LIN {X 0,Y 162.657,Z 541.681,A -85,B 0,C 180,E1 -31313.823,E2 -31313.823} C_VEL
LIN {X 0,Y 162.251,Z 555.226,A -85,B 0,C 180,E1 -31317.216,E2 -31317.216} C_VEL
LIN {X 0,Y 162.332,Z 566.74,A -85,B 0,C 180,E1 -31320.617,E2 -31320.617} C_VEL
LIN {X 0,Y 162.635,Z 577.197,A -85,B 0,C 180,E1 -31324.322,E2 -31324.322} C_VEL
LIN {X 0,Y 163.981,Z 589.038,A -85,B 0,C 180,E1 -31329.217,E2 -31329.217} C_VEL
LIN {X 0,Y 166.282,Z 597.77,A -85,B 0,C 180,E1 -31333.396,E2 -31333.396} C_VEL
LIN {X 0,Y 169.959,Z 606.171,A -85,B 0,C 180,E1 -31338.004,E2 -31338.004} C_VEL
LIN {X 0,Y 174.987,Z 613.199,A -85,B 0,C 180,E1 -31342.35,E2 -31342.35} C_VEL
LIN {X 0,Y 181.432,Z 619.004,A -85,B 0,C 180,E1 -31346.357,E2 -31346.357} C_VEL
LIN {X 0,Y 187.096,Z 622.568,A -85,B 0,C 180,E1 -31349.123,E2 -31349.123} C_VEL
LIN {X 0,Y 195.33,Z 626.257,A -85,B 0,C 180,E1 -31352.54,E2 -31352.54} C_VEL
LIN {X 0,Y 204.429,Z 628.796,A -85,B 0,C 180,E1 -31355.625,E2 -31355.625} C_VEL
LIN {X 0,Y 215.008,Z 630.267,A -85,B 0,C 180,E1 -31358.568,E2 -31358.568} C_VEL
LIN {X 0,Y 224.82,Z 630.463,A -85,B 0,C 180,E1 -31360.864,E2 -31360.864} C_VEL
LIN {X 0,Y 223.785,Z 630.854,A -85,B 0,C 180,E1 -31361.305,E2 -31361.305} C_VEL
LIN {X 0,Y 212.898,Z 633.183,A -85,B 0,C 180,E1 -31363.629,E2 -31363.629} C_VEL
LIN {X 0,Y 202.784,Z 634.608,A -85,B 0,C 180,E1 -31366.304,E2 -31366.304} C_VEL
LIN {X 0,Y 191.702,Z 635.182,A -85,B 0,C 180,E1 -31370.112,E2 -31370.112} C_VEL
LIN {X 0,Y 181.866,Z 634.463,A -85,B 0,C 180,E1 -31374.709,E2 -31374.709} C_VEL
LIN {X 0,Y 174.373,Z 632.741,A -85,B 0,C 180,E1 -31379.693,E2 -31379.693} C_VEL
LIN {X 0,Y 169.565,Z 638.187,A -85,B 0,C 180,E1 -31382.974,E2 -31382.974} C_VEL
LIN {X 0,Y 165.423,Z 642.984,A -85,B 0,C 180,E1 -31386.802,E2 -31386.802} C_VEL
LIN {X 0,Y 162.986,Z 645.969,A -85,B 0,C 180,E1 -31389.891,E2 -31389.891} C_VEL
LIN {X 0,Y 160.488,Z 649.343,A -85,B 0,C 180,E1 -31394.819,E2 -31394.819} C_VEL
LIN {X 0,Y 159.934,Z 650.447,A -85,B 0,C 180,E1 -31397.145,E2 -31397.145} C_VEL
LIN {X 0,Y 159.044,Z 651.219,A -85,B 0,C 180,E1 -31399.228,E2 -31399.228} C_VEL
LIN {X 0,Y 156.456,Z 651.707,A -85,B 0,C 180,E1 -31402.706,E2 -31402.706} C_VEL
LIN {X 0,Y 154.735,Z 651.565,A -85,B 0,C 180,E1 -31406.289,E2 -31406.289} C_VEL
LIN {X 0,Y 155.199,Z 651.263,A -85,B 0,C 180,E1 -31408.455,E2 -31408.455} C_VEL
LIN {X 0,Y 157.81,Z 650.765,A -85,B 0,C 180,E1 -31411.987,E2 -31411.987} C_VEL
LIN {X 0,Y 157.787,Z 658.681,A -85,B 0,C 180,E1 -31415.093,E2 -31415.093} C_VEL
LIN {X 0,Y 157.477,Z 665.759,A -85,B 0,C 180,E1 -31418.522,E2 -31418.522} C_VEL
LIN {X 0,Y 157.557,Z 673.281,A -85,B 0,C 180,E1 -31422.843,E2 -31422.843} C_VEL
LIN {X 0,Y 158.912,Z 680.871,A -85,B 0,C 180,E1 -31427.971,E2 -31427.971} C_VEL
LIN {X 0,Y 161.869,Z 687.258,A -85,B 0,C 180,E1 -31432.92,E2 -31432.92} C_VEL
LIN {X 0,Y 166.542,Z 692.636,A -85,B 0,C 180,E1 -31437.557,E2 -31437.557} C_VEL
LIN {X 0,Y 172.573,Z 696.952,A -85,B 0,C 180,E1 -31441.846,E2 -31441.846} C_VEL
LIN {X 0,Y 179.734,Z 700.291,A -85,B 0,C 180,E1 -31445.772,E2 -31445.772} C_VEL
LIN {X 0,Y 188.2,Z 702.78,A -85,B 0,C 180,E1 -31449.25,E2 -31449.25} C_VEL
LIN {X 0,Y 197.682,Z 704.359,A -85,B 0,C 180,E1 -31452.316,E2 -31452.316} C_VEL
LIN {X 0,Y 207.92,Z 704.957,A -85,B 0,C 180,E1 -31455.028,E2 -31455.028} C_VEL
LIN {X 0,Y 197.945,Z 704.33,A -85,B 0,C 180,E1 -31457.753,E2 -31457.753} C_VEL
LIN {X 0,Y 188.578,Z 702.73,A -85,B 0,C 180,E1 -31460.844,E2 -31460.844} C_VEL
LIN {X 0,Y 180.062,Z 700.21,A -85,B 0,C 180,E1 -31464.303,E2 -31464.303} C_VEL
LIN {X 0,Y 172.782,Z 696.814,A -85,B 0,C 180,E1 -31468.197,E2 -31468.197} C_VEL
LIN {X 0,Y 165.469,Z 691.187,A -85,B 0,C 180,E1 -31473.611,E2 -31473.611} C_VEL
LIN {X 0,Y 161.091,Z 685.52,A -85,B 0,C 180,E1 -31478.31,E2 -31478.31} C_VEL
LIN {X 0,Y 158.325,Z 678.763,A -85,B 0,C 180,E1 -31483.288,E2 -31483.288} C_VEL
LIN {X 0,Y 157.225,Z 669.662,A -85,B 0,C 180,E1 -31489.086,E2 -31489.086} C_VEL
LIN {X 0,Y 157.41,Z 661.083,A -85,B 0,C 180,E1 -31493.614,E2 -31493.614} C_VEL
LIN {X 0,Y 157.623,Z 653.684,A -85,B 0,C 180,E1 -31496.816,E2 -31496.816} C_VEL
LIN {X 0,Y 157.444,Z 644.543,A -85,B 0,C 180,E1 -31500.001,E2 -31500.001} C_VEL
LIN {X 0,Y 157.364,Z 633.619,A -85,B 0,C 180,E1 -31503.19,E2 -31503.19} C_VEL
LIN {X 0,Y 157.453,Z 620.345,A -85,B 0,C 180,E1 -31506.386,E2 -31506.386} C_VEL
LIN {X 0,Y 157.743,Z 605.275,A -85,B 0,C 180,E1 -31509.264,E2 -31509.264} C_VEL
LIN {X 0,Y 158.123,Z 591.449,A -85,B 0,C 180,E1 -31511.364,E2 -31511.364} C_VEL
LIN {X 0,Y 158.427,Z 575.605,A -85,B 0,C 180,E1 -31513.178,E2 -31513.178} C_VEL
LIN {X 0,Y 159.069,Z 531.92,A -85,B 0,C 180,E1 -31517.292,E2 -31517.292} C_VEL
LIN {X 0,Y 160.564,Z 481.479,A -85,B 0,C 180,E1 -31521.892,E2 -31521.892} C_VEL
LIN {X 0,Y 158.603,Z 451.78,A -85,B 0,C 180,E1 -31524.372,E2 -31524.372} C_VEL
LIN {X 0,Y 158.469,Z 439.257,A -85,B 0,C 180,E1 -31525.529,E2 -31525.529} C_VEL
LIN {X 0,Y 161.863,Z 413.266,A -85,B 0,C 180,E1 -31532.747,E2 -31532.747} C_VEL
LIN {X 0,Y 160.879,Z 408.168,A -85,B 0,C 180,E1 -31534.185,E2 -31534.185} C_VEL
LIN {X 0,Y 161.476,Z 409.866,A -85,B 0,C 180,E1 -31534.704,E2 -31534.704} C_VEL
LIN {X 0,Y 162.33,Z 410.505,A -85,B 0,C 180,E1 -31535.249,E2 -31535.249} C_VEL
LIN {X 0,Y 164.016,Z 410.046,A -85,B 0,C 180,E1 -31536.149,E2 -31536.149} C_VEL
LIN {X 0,Y 165.523,Z 408.754,A -85,B 0,C 180,E1 -31536.852,E2 -31536.852} C_VEL
LIN {X 0,Y 169.339,Z 408.335,A -85,B 0,C 180,E1 -31538.729,E2 -31538.729} C_VEL
LIN {X 0,Y 171.509,Z 407.086,A -85,B 0,C 180,E1 -31539.653,E2 -31539.653} C_VEL
LIN {X 0,Y 175.345,Z 406.759,A -85,B 0,C 180,E1 -31541.309,E2 -31541.309} C_VEL
LIN {X 0,Y 180.627,Z 415.01,A -85,B 0,C 180,E1 -31543.911,E2 -31543.911} C_VEL
LIN {X 0,Y 186.581,Z 425.308,A -85,B 0,C 180,E1 -31546.581,E2 -31546.581} C_VEL
LIN {X 0,Y 192.729,Z 437.493,A -85,B 0,C 180,E1 -31549.124,E2 -31549.124} C_VEL
LIN {X 0,Y 194.185,Z 440.713,A -85,B 0,C 180,E1 -31549.703,E2 -31549.703} C_VEL
LIN {X 0,Y 191.472,Z 490.951,A -85,B 0,C 180,E1 -31551.492,E2 -31551.492} C_VEL
LIN {X 0,Y 190.329,Z 504.695,A -85,B 0,C 180,E1 -31552.278,E2 -31552.278} C_VEL
LIN {X 0,Y 188.23,Z 519.107,A -85,B 0,C 180,E1 -31553.46,E2 -31553.46} C_VEL
LIN {X 0,Y 185.58,Z 531.813,A -85,B 0,C 180,E1 -31554.859,E2 -31554.859} C_VEL
LIN {X 0,Y 182.689,Z 543.452,A -85,B 0,C 180,E1 -31556.554,E2 -31556.554} C_VEL
LIN {X 0,Y 179.123,Z 555.581,A -85,B 0,C 180,E1 -31558.793,E2 -31558.793} C_VEL
LIN {X 0,Y 175.219,Z 566.598,A -85,B 0,C 180,E1 -31561.334,E2 -31561.334} C_VEL
LIN {X 0,Y 170.85,Z 577.269,A -85,B 0,C 180,E1 -31564.434,E2 -31564.434} C_VEL
LIN {X 0,Y 166.886,Z 586.379,A -85,B 0,C 180,E1 -31567.806,E2 -31567.806} C_VEL
LIN {X 0,Y 163.004,Z 594.923,A -85,B 0,C 180,E1 -31571.848,E2 -31571.848} C_VEL
LIN {X 0,Y 159.652,Z 601.853,A -85,B 0,C 180,E1 -31576.037,E2 -31576.037} C_VEL
LIN {X 0,Y 156.764,Z 608.082,A -85,B 0,C 180,E1 -31581.003,E2 -31581.003} C_VEL
LIN {X 0,Y 155.173,Z 611.678,A -85,B 0,C 180,E1 -31584.821,E2 -31584.821} C_VEL
LIN {X 0,Y 154.059,Z 615.204,A -85,B 0,C 180,E1 -31590,E2 -31590} C_VEL
LIN {X 0,Y 153.894,Z 617.381,A -85,B 0,C 180,E1 -31595.223,E2 -31595.223} C_VEL
LIN {X 0,Y 154.588,Z 618.271,A -85,B 0,C 180,E1 -31600.443,E2 -31600.443} C_VEL
LIN {X 0,Y 156.181,Z 617.88,A -85,B 0,C 180,E1 -31605.611,E2 -31605.611} C_VEL
LIN {X 0,Y 158.917,Z 616.168,A -85,B 0,C 180,E1 -31610.648,E2 -31610.648} C_VEL
LIN {X 0,Y 162.647,Z 613.091,A -85,B 0,C 180,E1 -31615.51,E2 -31615.51} C_VEL
LIN {X 0,Y 167.258,Z 608.524,A -85,B 0,C 180,E1 -31620.169,E2 -31620.169} C_VEL
LIN {X 0,Y 172.76,Z 602.335,A -85,B 0,C 180,E1 -31624.585,E2 -31624.585} C_VEL
LIN {X 0,Y 177.961,Z 595.766,A -85,B 0,C 180,E1 -31628.075,E2 -31628.075} C_VEL
LIN {X 0,Y 183.455,Z 588.119,A -85,B 0,C 180,E1 -31631.195,E2 -31631.195} C_VEL
LIN {X 0,Y 189.122,Z 579.325,A -85,B 0,C 180,E1 -31633.983,E2 -31633.983} C_VEL
LIN {X 0,Y 194.653,Z 569.152,A -85,B 0,C 180,E1 -31636.583,E2 -31636.583} C_VEL
LIN {X 0,Y 200.076,Z 557.787,A -85,B 0,C 180,E1 -31638.825,E2 -31638.825} C_VEL
LIN {X 0,Y 204.966,Z 545.823,A -85,B 0,C 180,E1 -31640.641,E2 -31640.641} C_VEL
LIN {X 0,Y 208.697,Z 534.273,A -85,B 0,C 180,E1 -31642.067,E2 -31642.067} C_VEL
LIN {X 0,Y 212.105,Z 520.79,A -85,B 0,C 180,E1 -31643.373,E2 -31643.373} C_VEL
LIN {X 0,Y 214.577,Z 507.153,A -85,B 0,C 180,E1 -31644.357,E2 -31644.357} C_VEL
LIN {X 0,Y 216.23,Z 493.322,A -85,B 0,C 180,E1 -31645.033,E2 -31645.033} C_VEL
LIN {X 0,Y 218.184,Z 463.682,A -85,B 0,C 180,E1 -31646.002,E2 -31646.002} C_VEL
LIN {X 0,Y 212.944,Z 453.225,A -85,B 0,C 180,E1 -31648.622,E2 -31648.622} C_VEL
LIN {X 0,Y 210.989,Z 449.575,A -85,B 0,C 180,E1 -31649.667,E2 -31649.667} C_VEL
LIN {X 0,Y 206.99,Z 459.803,A -85,B 0,C 180,E1 -31650.788,E2 -31650.788} C_VEL
LIN {X 0,Y 203.4,Z 466.877,A -85,B 0,C 180,E1 -31652.013,E2 -31652.013} C_VEL
LIN {X 0,Y 202.486,Z 468.575,A -85,B 0,C 180,E1 -31652.347,E2 -31652.347} C_VEL
LIN {X 0,Y 198.679,Z 481.103,A -85,B 0,C 180,E1 -31653.401,E2 -31653.401} C_VEL
LIN {X 0,Y 195.565,Z 489.455,A -85,B 0,C 180,E1 -31654.47,E2 -31654.47} C_VEL
LIN {X 0,Y 192.222,Z 496.043,A -85,B 0,C 180,E1 -31655.863,E2 -31655.863} C_VEL
LIN {X 0,Y 191.222,Z 497.747,A -85,B 0,C 180,E1 -31656.313,E2 -31656.313} C_VEL
LIN {X 0,Y 187.469,Z 508.563,A -85,B 0,C 180,E1 -31657.322,E2 -31657.322} C_VEL
LIN {X 0,Y 184.183,Z 515.642,A -85,B 0,C 180,E1 -31658.308,E2 -31658.308} C_VEL
LIN {X 0,Y 180.852,Z 521.347,A -85,B 0,C 180,E1 -31659.525,E2 -31659.525} C_VEL
LIN {X 0,Y 178.031,Z 525.18,A -85,B 0,C 180,E1 -31660.781,E2 -31660.781} C_VEL
LIN {X 0,Y 175.796,Z 527.75,A -85,B 0,C 180,E1 -31662.013,E2 -31662.013} C_VEL
LIN {X 0,Y 171.998,Z 533.916,A -85,B 0,C 180,E1 -31663.436,E2 -31663.436} C_VEL
LIN {X 0,Y 168.996,Z 537.903,A -85,B 0,C 180,E1 -31664.986,E2 -31664.986} C_VEL
LIN {X 0,Y 168.114,Z 538.939,A -85,B 0,C 180,E1 -31665.522,E2 -31665.522} C_VEL
LIN {X 0,Y 166.791,Z 540.084,A -85,B 0,C 180,E1 -31666.645,E2 -31666.645} C_VEL
LIN {X 0,Y 165.194,Z 542.014,A -85,B 0,C 180,E1 -31667.759,E2 -31667.759} C_VEL
LIN {X 0,Y 162.353,Z 546.074,A -85,B 0,C 180,E1 -31669.371,E2 -31669.371} C_VEL
LIN {X 0,Y 161.493,Z 547.163,A -85,B 0,C 180,E1 -31670.008,E2 -31670.008} C_VEL
LIN {X 0,Y 160.015,Z 548.819,A -85,B 0,C 180,E1 -31671.509,E2 -31671.509} C_VEL
LIN {X 0,Y 159.456,Z 549.259,A -85,B 0,C 180,E1 -31672.427,E2 -31672.427} C_VEL
LIN {X 0,Y 158.404,Z 550.699,A -85,B 0,C 180,E1 -31673.472,E2 -31673.472} C_VEL
LIN {X 0,Y 156.612,Z 553.438,A -85,B 0,C 180,E1 -31674.867,E2 -31674.867} C_VEL
LIN {X 0,Y 155.163,Z 555.396,A -85,B 0,C 180,E1 -31677.412,E2 -31677.412} C_VEL
LIN {X 0,Y 155.611,Z 554.521,A -85,B 0,C 180,E1 -31678.145,E2 -31678.145} C_VEL
LIN {X 0,Y 155.791,Z 566.718,A -85,B 0,C 180,E1 -31681.932,E2 -31681.932} C_VEL
LIN {X 0,Y 156.222,Z 577.22,A -85,B 0,C 180,E1 -31685.789,E2 -31685.789} C_VEL
LIN {X 0,Y 157.591,Z 587.719,A -85,B 0,C 180,E1 -31690.24,E2 -31690.24} C_VEL
LIN {X 0,Y 160.433,Z 597.884,A -85,B 0,C 180,E1 -31695.186,E2 -31695.186} C_VEL
LIN {X 0,Y 164.519,Z 606.427,A -85,B 0,C 180,E1 -31699.913,E2 -31699.913} C_VEL
LIN {X 0,Y 170.034,Z 613.597,A -85,B 0,C 180,E1 -31704.326,E2 -31704.326} C_VEL
LIN {X 0,Y 176.988,Z 619.531,A -85,B 0,C 180,E1 -31708.353,E2 -31708.353} C_VEL
LIN {X 0,Y 185.041,Z 624.272,A -85,B 0,C 180,E1 -31712.001,E2 -31712.001} C_VEL
LIN {X 0,Y 193.935,Z 627.835,A -85,B 0,C 180,E1 -31715.301,E2 -31715.301} C_VEL
LIN {X 0,Y 203.649,Z 630.282,A -85,B 0,C 180,E1 -31718.25,E2 -31718.25} C_VEL
LIN {X 0,Y 214.07,Z 631.593,A -85,B 0,C 180,E1 -31720.874,E2 -31720.874} C_VEL
LIN {X 0,Y 202.802,Z 633.121,A -85,B 0,C 180,E1 -31723.505,E2 -31723.505} C_VEL
LIN {X 0,Y 193.017,Z 633.7,A -85,B 0,C 180,E1 -31726.409,E2 -31726.409} C_VEL
LIN {X 0,Y 184.09,Z 633.471,A -85,B 0,C 180,E1 -31729.696,E2 -31729.696} C_VEL
LIN {X 0,Y 176.353,Z 632.473,A -85,B 0,C 180,E1 -31733.432,E2 -31733.432} C_VEL
LIN {X 0,Y 169.681,Z 630.635,A -85,B 0,C 180,E1 -31737.719,E2 -31737.719} C_VEL
LIN {X 0,Y 164.746,Z 635.91,A -85,B 0,C 180,E1 -31740.728,E2 -31740.728} C_VEL
LIN {X 0,Y 159.345,Z 641.81,A -85,B 0,C 180,E1 -31745.316,E2 -31745.316} C_VEL
LIN {X 0,Y 156.322,Z 645.271,A -85,B 0,C 180,E1 -31748.994,E2 -31748.994} C_VEL
LIN {X 0,Y 153.612,Z 648.614,A -85,B 0,C 180,E1 -31754.121,E2 -31754.121} C_VEL
LIN {X 0,Y 152.65,Z 650.665,A -85,B 0,C 180,E1 -31759.423,E2 -31759.423} C_VEL
LIN {X 0,Y 153.514,Z 651.473,A -85,B 0,C 180,E1 -31764.764,E2 -31764.764} C_VEL
LIN {X 0,Y 155.199,Z 651.263,A -85,B 0,C 180,E1 -31768.455,E2 -31768.455} C_VEL
LIN {X 0,Y 155.419,Z 651.231,A -85,B 0,C 180,E1 -31769.945,E2 -31769.945} C_VEL
LIN {X 0,Y 154.353,Z 651.761,A -85,B 0,C 180,E1 -31771.92,E2 -31771.92} C_VEL
LIN {X 0,Y 152.381,Z 653.626,A -85,B 0,C 180,E1 -31774.307,E2 -31774.307} C_VEL
LIN {X 0,Y 151.566,Z 656.014,A -85,B 0,C 180,E1 -31775.853,E2 -31775.853} C_VEL
LIN {X 0,Y 151.539,Z 656.445,A -85,B 0,C 180,E1 -31776.056,E2 -31776.056} C_VEL
LIN {X 0,Y 151.241,Z 664.317,A -85,B 0,C 180,E1 -31780.007,E2 -31780.007} C_VEL
LIN {X 0,Y 151.502,Z 672.172,A -85,B 0,C 180,E1 -31784.729,E2 -31784.729} C_VEL
LIN {X 0,Y 153.324,Z 679.816,A -85,B 0,C 180,E1 -31790.037,E2 -31790.037} C_VEL
LIN {X 0,Y 156.863,Z 686.286,A -85,B 0,C 180,E1 -31795.1,E2 -31795.1} C_VEL
LIN {X 0,Y 163.537,Z 692.953,A -85,B 0,C 180,E1 -31800.928,E2 -31800.928} C_VEL
LIN {X 0,Y 170.251,Z 697.118,A -85,B 0,C 180,E1 -31805.168,E2 -31805.168} C_VEL
LIN {X 0,Y 178.347,Z 700.403,A -85,B 0,C 180,E1 -31808.931,E2 -31808.931} C_VEL
LIN {X 0,Y 187.535,Z 702.822,A -85,B 0,C 180,E1 -31812.245,E2 -31812.245} C_VEL
LIN {X 0,Y 196.063,Z 704.167,A -85,B 0,C 180,E1 -31814.714,E2 -31814.714} C_VEL
LIN {X 0,Y 196.183,Z 704.175,A -85,B 0,C 180,E1 -31815.4,E2 -31815.4} C_VEL
LIN {X 0,Y 187.854,Z 702.823,A -85,B 0,C 180,E1 -31817.844,E2 -31817.844} C_VEL
LIN {X 0,Y 178.719,Z 700.391,A -85,B 0,C 180,E1 -31821.166,E2 -31821.166} C_VEL
LIN {X 0,Y 170.545,Z 697.061,A -85,B 0,C 180,E1 -31824.902,E2 -31824.902} C_VEL
LIN {X 0,Y 162.239,Z 691.601,A -85,B 0,C 180,E1 -31830.232,E2 -31830.232} C_VEL
LIN {X 0,Y 156.953,Z 686.096,A -85,B 0,C 180,E1 -31834.916,E2 -31834.916} C_VEL
LIN {X 0,Y 153.359,Z 679.585,A -85,B 0,C 180,E1 -31839.968,E2 -31839.968} C_VEL
LIN {X 0,Y 151.254,Z 670.783,A -85,B 0,C 180,E1 -31845.93,E2 -31845.93} C_VEL
LIN {X 0,Y 150.98,Z 663.176,A -85,B 0,C 180,E1 -31850.399,E2 -31850.399} C_VEL
LIN {X 0,Y 151.298,Z 655.902,A -85,B 0,C 180,E1 -31854.022,E2 -31854.022} C_VEL
LIN {X 0,Y 151.271,Z 647.634,A -85,B 0,C 180,E1 -31857.347,E2 -31857.347} C_VEL
LIN {X 0,Y 150.99,Z 636.4,A -85,B 0,C 180,E1 -31860.997,E2 -31860.997} C_VEL
LIN {X 0,Y 150.9,Z 625.256,A -85,B 0,C 180,E1 -31863.993,E2 -31863.993} C_VEL
LIN {X 0,Y 150.979,Z 613.352,A -85,B 0,C 180,E1 -31866.661,E2 -31866.661} C_VEL
LIN {X 0,Y 151.311,Z 597.765,A -85,B 0,C 180,E1 -31869.493,E2 -31869.493} C_VEL
LIN {X 0,Y 151.633,Z 582.224,A -85,B 0,C 180,E1 -31871.611,E2 -31871.611} C_VEL
LIN {X 0,Y 151.969,Z 551.348,A -85,B 0,C 180,E1 -31874.77,E2 -31874.77} C_VEL
LIN {X 0,Y 153.545,Z 481.43,A -85,B 0,C 180,E1 -31881.54,E2 -31881.54} C_VEL
LIN {X 0,Y 151.664,Z 454.367,A -85,B 0,C 180,E1 -31883.916,E2 -31883.916} C_VEL
LIN {X 0,Y 151.387,Z 439.32,A -85,B 0,C 180,E1 -31885.341,E2 -31885.341} C_VEL
LIN {X 0,Y 153.472,Z 421.408,A -85,B 0,C 180,E1 -31890.562,E2 -31890.562} C_VEL
LIN {X 0,Y 153.625,Z 423.294,A -85,B 0,C 180,E1 -31890.861,E2 -31890.861} C_VEL
LIN {X 0,Y 154.383,Z 423.859,A -85,B 0,C 180,E1 -31891.451,E2 -31891.451} C_VEL
LIN {X 0,Y 155.936,Z 423.038,A -85,B 0,C 180,E1 -31892.427,E2 -31892.427} C_VEL
LIN {X 0,Y 158.972,Z 419.477,A -85,B 0,C 180,E1 -31894.033,E2 -31894.033} C_VEL
LIN {X 0,Y 160.226,Z 417.725,A -85,B 0,C 180,E1 -31894.633,E2 -31894.633} C_VEL
LIN {X 0,Y 163.793,Z 417.114,A -85,B 0,C 180,E1 -31896.587,E2 -31896.587} C_VEL
LIN {X 0,Y 166.051,Z 415.745,A -85,B 0,C 180,E1 -31897.657,E2 -31897.657} C_VEL
LIN {X 0,Y 169.81,Z 415.105,A -85,B 0,C 180,E1 -31899.433,E2 -31899.433} C_VEL
LIN {X 0,Y 171.695,Z 414.098,A -85,B 0,C 180,E1 -31900.221,E2 -31900.221} C_VEL
LIN {X 0,Y 173.406,Z 414.308,A -85,B 0,C 180,E1 -31900.984,E2 -31900.984} C_VEL
LIN {X 0,Y 178.841,Z 423.278,A -85,B 0,C 180,E1 -31903.742,E2 -31903.742} C_VEL
LIN {X 0,Y 184.373,Z 433.486,A -85,B 0,C 180,E1 -31906.305,E2 -31906.305} C_VEL
LIN {X 0,Y 188.9,Z 442.948,A -85,B 0,C 180,E1 -31908.267,E2 -31908.267} C_VEL
LIN {X 0,Y 186.027,Z 494.794,A -85,B 0,C 180,E1 -31910.201,E2 -31910.201} C_VEL
LIN {X 0,Y 184.475,Z 509.247,A -85,B 0,C 180,E1 -31911.121,E2 -31911.121} C_VEL
LIN {X 0,Y 182.212,Z 523.042,A -85,B 0,C 180,E1 -31912.392,E2 -31912.392} C_VEL
LIN {X 0,Y 178.999,Z 536.78,A -85,B 0,C 180,E1 -31914.058,E2 -31914.058} C_VEL
LIN {X 0,Y 175.608,Z 549.043,A -85,B 0,C 180,E1 -31916.054,E2 -31916.054} C_VEL
LIN {X 0,Y 171.506,Z 561.419,A -85,B 0,C 180,E1 -31918.62,E2 -31918.62} C_VEL
LIN {X 0,Y 167.49,Z 571.571,A -85,B 0,C 180,E1 -31921.254,E2 -31921.254} C_VEL
LIN {X 0,Y 163.037,Z 581.692,A -85,B 0,C 180,E1 -31924.557,E2 -31924.557} C_VEL
LIN {X 0,Y 159.161,Z 590.046,A -85,B 0,C 180,E1 -31928.033,E2 -31928.033} C_VEL
LIN {X 0,Y 155.251,Z 598.039,A -85,B 0,C 180,E1 -31932.27,E2 -31932.27} C_VEL
LIN {X 0,Y 151.951,Z 604.506,A -85,B 0,C 180,E1 -31936.675,E2 -31936.675} C_VEL
LIN {X 0,Y 149.172,Z 610.251,A -85,B 0,C 180,E1 -31941.902,E2 -31941.902} C_VEL
LIN {X 0,Y 147.419,Z 614.468,A -85,B 0,C 180,E1 -31947.277,E2 -31947.277} C_VEL
LIN {X 0,Y 146.81,Z 617.276,A -85,B 0,C 180,E1 -31952.735,E2 -31952.735} C_VEL
LIN {X 0,Y 147.115,Z 618.779,A -85,B 0,C 180,E1 -31958.212,E2 -31958.212} C_VEL
LIN {X 0,Y 148.378,Z 618.998,A -85,B 0,C 180,E1 -31963.653,E2 -31963.653} C_VEL
LIN {X 0,Y 150.617,Z 617.932,A -85,B 0,C 180,E1 -31968.999,E2 -31968.999} C_VEL
LIN {X 0,Y 154.175,Z 615.504,A -85,B 0,C 180,E1 -31974.135,E2 -31974.135} C_VEL
LIN {X 0,Y 158.572,Z 611.66,A -85,B 0,C 180,E1 -31979.072,E2 -31979.072} C_VEL
LIN {X 0,Y 163.956,Z 606.263,A -85,B 0,C 180,E1 -31983.737,E2 -31983.737} C_VEL
LIN {X 0,Y 168.593,Z 601.122,A -85,B 0,C 180,E1 -31987.044,E2 -31987.044} C_VEL
LIN {X 0,Y 174.478,Z 593.686,A -85,B 0,C 180,E1 -31990.72,E2 -31990.72} C_VEL
LIN {X 0,Y 180.068,Z 585.893,A -85,B 0,C 180,E1 -31993.667,E2 -31993.667} C_VEL
LIN {X 0,Y 186.09,Z 576.453,A -85,B 0,C 180,E1 -31996.434,E2 -31996.434} C_VEL
LIN {X 0,Y 191.37,Z 566.582,A -85,B 0,C 180,E1 -31998.789,E2 -31998.789} C_VEL
LIN {X 0,Y 196.58,Z 555.608,A -85,B 0,C 180,E1 -32000.805,E2 -32000.805} C_VEL
LIN {X 0,Y 201.646,Z 542.888,A -85,B 0,C 180,E1 -32002.618,E2 -32002.618} C_VEL
LIN {X 0,Y 205.502,Z 530.416,A -85,B 0,C 180,E1 -32004.049,E2 -32004.049} C_VEL
LIN {X 0,Y 208.593,Z 517.3,A -85,B 0,C 180,E1 -32005.219,E2 -32005.219} C_VEL
LIN {X 0,Y 211.028,Z 502.908,A -85,B 0,C 180,E1 -32006.142,E2 -32006.142} C_VEL
LIN {X 0,Y 212.464,Z 487.742,A -85,B 0,C 180,E1 -32006.78,E2 -32006.78} C_VEL
LIN {X 0,Y 213.912,Z 466.76,A -85,B 0,C 180,E1 -32007.434,E2 -32007.434} C_VEL
LIN {X 0,Y 211.108,Z 460.966,A -85,B 0,C 180,E1 -32008.911,E2 -32008.911} C_VEL
LIN {X 0,Y 210.862,Z 461.043,A -85,B 0,C 180,E1 -32009.01,E2 -32009.01} C_VEL
LIN {X 0,Y 207.215,Z 468.684,A -85,B 0,C 180,E1 -32010.108,E2 -32010.108} C_VEL
LIN {X 0,Y 205.195,Z 472.414,A -85,B 0,C 180,E1 -32010.782,E2 -32010.782} C_VEL
LIN {X 0,Y 201.311,Z 484.635,A -85,B 0,C 180,E1 -32011.802,E2 -32011.802} C_VEL
LIN {X 0,Y 198.001,Z 493.168,A -85,B 0,C 180,E1 -32012.855,E2 -32012.855} C_VEL
LIN {X 0,Y 194.286,Z 500.159,A -85,B 0,C 180,E1 -32014.225,E2 -32014.225} C_VEL
LIN {X 0,Y 193.243,Z 501.915,A -85,B 0,C 180,E1 -32014.609,E2 -32014.609} C_VEL
LIN {X 0,Y 189.246,Z 512.081,A -85,B 0,C 180,E1 -32015.532,E2 -32015.532} C_VEL
LIN {X 0,Y 185.524,Z 519.423,A -85,B 0,C 180,E1 -32016.497,E2 -32016.497} C_VEL
LIN {X 0,Y 181.712,Z 525.443,A -85,B 0,C 180,E1 -32017.689,E2 -32017.689} C_VEL
LIN {X 0,Y 177.821,Z 530.392,A -85,B 0,C 180,E1 -32019.236,E2 -32019.236} C_VEL
LIN {X 0,Y 176.528,Z 531.755,A -85,B 0,C 180,E1 -32019.861,E2 -32019.861} C_VEL
LIN {X 0,Y 175.135,Z 533.532,A -85,B 0,C 180,E1 -32020.45,E2 -32020.45} C_VEL
LIN {X 0,Y 171.819,Z 538.312,A -85,B 0,C 180,E1 -32021.582,E2 -32021.582} C_VEL
LIN {X 0,Y 168.298,Z 542.641,A -85,B 0,C 180,E1 -32023.187,E2 -32023.187} C_VEL
LIN {X 0,Y 166.725,Z 544.338,A -85,B 0,C 180,E1 -32024.027,E2 -32024.027} C_VEL
LIN {X 0,Y 164.224,Z 546.612,A -85,B 0,C 180,E1 -32025.803,E2 -32025.803} C_VEL
LIN {X 0,Y 160.173,Z 551.654,A -85,B 0,C 180,E1 -32028.011,E2 -32028.011} C_VEL
LIN {X 0,Y 157.981,Z 553.968,A -85,B 0,C 180,E1 -32029.784,E2 -32029.784} C_VEL
LIN {X 0,Y 156.876,Z 555.018,A -85,B 0,C 180,E1 -32031.009,E2 -32031.009} C_VEL
LIN {X 0,Y 155.513,Z 556.648,A -85,B 0,C 180,E1 -32032.269,E2 -32032.269} C_VEL
LIN {X 0,Y 153.915,Z 558.774,A -85,B 0,C 180,E1 -32033.465,E2 -32033.465} C_VEL
LIN {X 0,Y 152.952,Z 559.885,A -85,B 0,C 180,E1 -32034.744,E2 -32034.744} C_VEL
LIN {X 0,Y 151.612,Z 561.531,A -85,B 0,C 180,E1 -32037.351,E2 -32037.351} C_VEL
LIN {X 0,Y 150.242,Z 563.695,A -85,B 0,C 180,E1 -32038.664,E2 -32038.664} C_VEL
LIN {X 0,Y 149.259,Z 565.345,A -85,B 0,C 180,E1 -32039.999,E2 -32039.999} C_VEL
LIN {X 0,Y 148.931,Z 566.385,A -85,B 0,C 180,E1 -32042.695,E2 -32042.695} C_VEL
LIN {X 0,Y 149.326,Z 565.929,A -85,B 0,C 180,E1 -32043.108,E2 -32043.108} C_VEL
LIN {X 0,Y 149.923,Z 577.167,A -85,B 0,C 180,E1 -32047.381,E2 -32047.381} C_VEL
LIN {X 0,Y 151.95,Z 589.051,A -85,B 0,C 180,E1 -32052.647,E2 -32052.647} C_VEL
LIN {X 0,Y 154.833,Z 597.94,A -85,B 0,C 180,E1 -32057.1,E2 -32057.1} C_VEL
LIN {X 0,Y 159.331,Z 606.551,A -85,B 0,C 180,E1 -32061.942,E2 -32061.942} C_VEL
LIN {X 0,Y 165.337,Z 613.866,A -85,B 0,C 180,E1 -32066.412,E2 -32066.412} C_VEL
LIN {X 0,Y 172.794,Z 619.97,A -85,B 0,C 180,E1 -32070.444,E2 -32070.444} C_VEL
LIN {X 0,Y 181.238,Z 624.845,A -85,B 0,C 180,E1 -32074.082,E2 -32074.082} C_VEL
LIN {X 0,Y 188.164,Z 627.757,A -85,B 0,C 180,E1 -32076.555,E2 -32076.555} C_VEL
LIN {X 0,Y 198.103,Z 630.673,A -85,B 0,C 180,E1 -32079.526,E2 -32079.526} C_VEL
LIN {X 0,Y 202.451,Z 631.561,A -85,B 0,C 180,E1 -32080.646,E2 -32080.646} C_VEL
LIN {X 0,Y 201.668,Z 631.797,A -85,B 0,C 180,E1 -32081.161,E2 -32081.161} C_VEL
LIN {X 0,Y 192.914,Z 632.212,A -85,B 0,C 180,E1 -32083.433,E2 -32083.433} C_VEL
LIN {X 0,Y 183.324,Z 632.04,A -85,B 0,C 180,E1 -32086.547,E2 -32086.547} C_VEL
LIN {X 0,Y 174.823,Z 631.076,A -85,B 0,C 180,E1 -32090.129,E2 -32090.129} C_VEL
LIN {X 0,Y 165.127,Z 628.65,A -85,B 0,C 180,E1 -32095.71,E2 -32095.71} C_VEL
LIN {X 0,Y 160.24,Z 633.557,A -85,B 0,C 180,E1 -32098.362,E2 -32098.362} C_VEL
LIN {X 0,Y 154.185,Z 639.854,A -85,B 0,C 180,E1 -32102.98,E2 -32102.98} C_VEL
LIN {X 0,Y 149.697,Z 644.572,A -85,B 0,C 180,E1 -32108.017,E2 -32108.017} C_VEL
LIN {X 0,Y 146.763,Z 647.886,A -85,B 0,C 180,E1 -32113.36,E2 -32113.36} C_VEL
LIN {X 0,Y 145.604,Z 649.905,A -85,B 0,C 180,E1 -32118.905,E2 -32118.905} C_VEL
LIN {X 0,Y 146.348,Z 650.683,A -85,B 0,C 180,E1 -32124.507,E2 -32124.507} C_VEL
LIN {X 0,Y 148.949,Z 650.224,A -85,B 0,C 180,E1 -32130,E2 -32130} C_VEL
LIN {X 0,Y 151.539,Z 649.504,A -85,B 0,C 180,E1 -32133.229,E2 -32133.229} C_VEL
LIN {X 0,Y 151.539,Z 656.445,A -85,B 0,C 180,E1 -32136.056,E2 -32136.056} C_VEL
LIN {X 0,Y 150.83,Z 659.852,A -85,B 0,C 180,E1 -32137.859,E2 -32137.859} C_VEL
LIN {X 0,Y 149.347,Z 662.591,A -85,B 0,C 180,E1 -32139.79,E2 -32139.79} C_VEL
LIN {X 0,Y 145.907,Z 668.14,A -85,B 0,C 180,E1 -32144.615,E2 -32144.615} C_VEL
LIN {X 0,Y 145.676,Z 670.842,A -85,B 0,C 180,E1 -32146.704,E2 -32146.704} C_VEL
LIN {X 0,Y 148.047,Z 678.646,A -85,B 0,C 180,E1 -32152.24,E2 -32152.24} C_VEL
LIN {X 0,Y 152.165,Z 685.224,A -85,B 0,C 180,E1 -32157.407,E2 -32157.407} C_VEL
LIN {X 0,Y 157.795,Z 690.749,A -85,B 0,C 180,E1 -32162.186,E2 -32162.186} C_VEL
LIN {X 0,Y 164.698,Z 695.298,A -85,B 0,C 180,E1 -32166.541,E2 -32166.541} C_VEL
LIN {X 0,Y 173.008,Z 698.96,A -85,B 0,C 180,E1 -32170.374,E2 -32170.374} C_VEL
LIN {X 0,Y 184.625,Z 702.278,A -85,B 0,C 180,E1 -32174.396,E2 -32174.396} C_VEL
LIN {X 0,Y 185.781,Z 702.533,A -85,B 0,C 180,E1 -32174.728,E2 -32174.728} C_VEL
LIN {X 0,Y 184.792,Z 702.304,A -85,B 0,C 180,E1 -32175.727,E2 -32175.727} C_VEL
LIN {X 0,Y 173.353,Z 698.99,A -85,B 0,C 180,E1 -32179.723,E2 -32179.723} C_VEL
LIN {X 0,Y 164.976,Z 695.268,A -85,B 0,C 180,E1 -32183.53,E2 -32183.53} C_VEL
LIN {X 0,Y 156.417,Z 689.386,A -85,B 0,C 180,E1 -32189.005,E2 -32189.005} C_VEL
LIN {X 0,Y 150.999,Z 683.514,A -85,B 0,C 180,E1 -32193.853,E2 -32193.853} C_VEL
LIN {X 0,Y 146.602,Z 674.722,A -85,B 0,C 180,E1 -32200.462,E2 -32200.462} C_VEL
LIN {X 0,Y 145.017,Z 664.813,A -85,B 0,C 180,E1 -32206.962,E2 -32206.962} C_VEL
LIN {X 0,Y 145.072,Z 654.835,A -85,B 0,C 180,E1 -32212.371,E2 -32212.371} C_VEL
LIN {X 0,Y 145.147,Z 648.525,A -85,B 0,C 180,E1 -32215.156,E2 -32215.156} C_VEL
LIN {X 0,Y 144.812,Z 638.852,A -85,B 0,C 180,E1 -32218.615,E2 -32218.615} C_VEL
LIN {X 0,Y 144.577,Z 627.133,A -85,B 0,C 180,E1 -32222.083,E2 -32222.083} C_VEL
LIN {X 0,Y 144.505,Z 615.8,A -85,B 0,C 180,E1 -32224.867,E2 -32224.867} C_VEL
LIN {X 0,Y 144.624,Z 601.859,A -85,B 0,C 180,E1 -32227.655,E2 -32227.655} C_VEL
LIN {X 0,Y 144.882,Z 587.536,A -85,B 0,C 180,E1 -32229.918,E2 -32229.918} C_VEL
LIN {X 0,Y 145.114,Z 569.012,A -85,B 0,C 180,E1 -32232.106,E2 -32232.106} C_VEL
LIN {X 0,Y 146.503,Z 481.147,A -85,B 0,C 180,E1 -32241.152,E2 -32241.152} C_VEL
LIN {X 0,Y 144.515,Z 452.075,A -85,B 0,C 180,E1 -32243.83,E2 -32243.83} C_VEL
LIN {X 0,Y 144.312,Z 440.609,A -85,B 0,C 180,E1 -32244.924,E2 -32244.924} C_VEL
LIN {X 0,Y 144.478,Z 443.309,A -85,B 0,C 180,E1 -32245.515,E2 -32245.515} C_VEL
LIN {X 0,Y 144.732,Z 443.793,A -85,B 0,C 180,E1 -32245.822,E2 -32245.822} C_VEL
LIN {X 0,Y 145.562,Z 443.205,A -85,B 0,C 180,E1 -32246.528,E2 -32246.528} C_VEL
LIN {X 0,Y 146.539,Z 441.471,A -85,B 0,C 180,E1 -32247.2,E2 -32247.2} C_VEL
LIN {X 0,Y 149.2,Z 437.654,A -85,B 0,C 180,E1 -32249.003,E2 -32249.003} C_VEL
LIN {X 0,Y 153.035,Z 430.819,A -85,B 0,C 180,E1 -32251.184,E2 -32251.184} C_VEL
LIN {X 0,Y 155.165,Z 430.47,A -85,B 0,C 180,E1 -32252.609,E2 -32252.609} C_VEL
LIN {X 0,Y 157.514,Z 428.678,A -85,B 0,C 180,E1 -32253.945,E2 -32253.945} C_VEL
LIN {X 0,Y 160.905,Z 424.716,A -85,B 0,C 180,E1 -32255.609,E2 -32255.609} C_VEL
LIN {X 0,Y 164.452,Z 423.779,A -85,B 0,C 180,E1 -32257.449,E2 -32257.449} C_VEL
LIN {X 0,Y 166.084,Z 422.815,A -85,B 0,C 180,E1 -32258.203,E2 -32258.203} C_VEL
LIN {X 0,Y 169.866,Z 422.052,A -85,B 0,C 180,E1 -32259.945,E2 -32259.945} C_VEL
LIN {X 0,Y 171.354,Z 421.609,A -85,B 0,C 180,E1 -32260.582,E2 -32260.582} C_VEL
LIN {X 0,Y 177.78,Z 433.01,A -85,B 0,C 180,E1 -32263.934,E2 -32263.934} C_VEL
LIN {X 0,Y 183.808,Z 445.47,A -85,B 0,C 180,E1 -32266.788,E2 -32266.788} C_VEL
LIN {X 0,Y 180.907,Z 495.25,A -85,B 0,C 180,E1 -32268.675,E2 -32268.675} C_VEL
LIN {X 0,Y 179.31,Z 509.644,A -85,B 0,C 180,E1 -32269.594,E2 -32269.594} C_VEL
LIN {X 0,Y 176.954,Z 523.531,A -85,B 0,C 180,E1 -32270.887,E2 -32270.887} C_VEL
LIN {X 0,Y 173.851,Z 536.458,A -85,B 0,C 180,E1 -32272.455,E2 -32272.455} C_VEL
LIN {X 0,Y 170.269,Z 548.936,A -85,B 0,C 180,E1 -32274.475,E2 -32274.475} C_VEL
LIN {X 0,Y 166.432,Z 560.303,A -85,B 0,C 180,E1 -32276.831,E2 -32276.831} C_VEL
LIN {X 0,Y 162.202,Z 570.772,A -85,B 0,C 180,E1 -32279.509,E2 -32279.509} C_VEL
LIN {X 0,Y 157.376,Z 581.33,A -85,B 0,C 180,E1 -32282.93,E2 -32282.93} C_VEL
LIN {X 0,Y 153.335,Z 589.733,A -85,B 0,C 180,E1 -32286.441,E2 -32286.441} C_VEL
LIN {X 0,Y 149.685,Z 596.867,A -85,B 0,C 180,E1 -32290.169,E2 -32290.169} C_VEL
LIN {X 0,Y 146.003,Z 603.722,A -85,B 0,C 180,E1 -32294.701,E2 -32294.701} C_VEL
LIN {X 0,Y 142.838,Z 609.881,A -85,B 0,C 180,E1 -32300.118,E2 -32300.118} C_VEL
LIN {X 0,Y 141.14,Z 613.407,A -85,B 0,C 180,E1 -32304.304,E2 -32304.304} C_VEL
LIN {X 0,Y 139.956,Z 616.871,A -85,B 0,C 180,E1 -32310,E2 -32310} C_VEL
LIN {X 0,Y 139.817,Z 618.993,A -85,B 0,C 180,E1 -32315.751,E2 -32315.751} C_VEL
LIN {X 0,Y 140.659,Z 619.828,A -85,B 0,C 180,E1 -32321.49,E2 -32321.49} C_VEL
LIN {X 0,Y 142.54,Z 619.38,A -85,B 0,C 180,E1 -32327.149,E2 -32327.149} C_VEL
LIN {X 0,Y 145.722,Z 617.6,A -85,B 0,C 180,E1 -32332.616,E2 -32332.616} C_VEL
LIN {X 0,Y 149.944,Z 614.44,A -85,B 0,C 180,E1 -32337.849,E2 -32337.849} C_VEL
LIN {X 0,Y 155.139,Z 609.802,A -85,B 0,C 180,E1 -32342.807,E2 -32342.807} C_VEL
LIN {X 0,Y 161.256,Z 603.541,A -85,B 0,C 180,E1 -32347.454,E2 -32347.454} C_VEL
LIN {X 0,Y 167.289,Z 596.532,A -85,B 0,C 180,E1 -32351.262,E2 -32351.262} C_VEL
LIN {X 0,Y 173.016,Z 589.156,A -85,B 0,C 180,E1 -32354.296,E2 -32354.296} C_VEL
LIN {X 0,Y 179.165,Z 580.26,A -85,B 0,C 180,E1 -32357.142,E2 -32357.142} C_VEL
LIN {X 0,Y 185.649,Z 569.08,A -85,B 0,C 180,E1 -32359.988,E2 -32359.988} C_VEL
LIN {X 0,Y 191.592,Z 557.178,A -85,B 0,C 180,E1 -32362.242,E2 -32362.242} C_VEL
LIN {X 0,Y 196.834,Z 544.639,A -85,B 0,C 180,E1 -32364.055,E2 -32364.055} C_VEL
LIN {X 0,Y 200.825,Z 532.423,A -85,B 0,C 180,E1 -32365.488,E2 -32365.488} C_VEL
LIN {X 0,Y 204.157,Z 519.113,A -85,B 0,C 180,E1 -32366.705,E2 -32366.705} C_VEL
LIN {X 0,Y 206.554,Z 505.958,A -85,B 0,C 180,E1 -32367.585,E2 -32367.585} C_VEL
LIN {X 0,Y 208.192,Z 491.526,A -85,B 0,C 180,E1 -32368.24,E2 -32368.24} C_VEL
LIN {X 0,Y 209.446,Z 473.815,A -85,B 0,C 180,E1 -32368.819,E2 -32368.819} C_VEL
LIN {X 0,Y 208.005,Z 476.322,A -85,B 0,C 180,E1 -32369.275,E2 -32369.275} C_VEL
LIN {X 0,Y 203.988,Z 488.471,A -85,B 0,C 180,E1 -32370.275,E2 -32370.275} C_VEL
LIN {X 0,Y 200.338,Z 497.257,A -85,B 0,C 180,E1 -32371.326,E2 -32371.326} C_VEL
LIN {X 0,Y 196.225,Z 504.439,A -85,B 0,C 180,E1 -32372.64,E2 -32372.64} C_VEL
LIN {X 0,Y 195.21,Z 506.221,A -85,B 0,C 180,E1 -32372.956,E2 -32372.956} C_VEL
LIN {X 0,Y 191.076,Z 515.617,A -85,B 0,C 180,E1 -32373.759,E2 -32373.759} C_VEL
LIN {X 0,Y 187.456,Z 522.314,A -85,B 0,C 180,E1 -32374.552,E2 -32374.552} C_VEL
LIN {X 0,Y 183.118,Z 528.817,A -85,B 0,C 180,E1 -32375.719,E2 -32375.719} C_VEL
LIN {X 0,Y 178.535,Z 534.474,A -85,B 0,C 180,E1 -32377.27,E2 -32377.27} C_VEL
LIN {X 0,Y 175.851,Z 537.2,A -85,B 0,C 180,E1 -32378.38,E2 -32378.38} C_VEL
LIN {X 0,Y 170.455,Z 544.048,A -85,B 0,C 180,E1 -32380.147,E2 -32380.147} C_VEL
LIN {X 0,Y 165.868,Z 548.988,A -85,B 0,C 180,E1 -32382.157,E2 -32382.157} C_VEL
LIN {X 0,Y 164.832,Z 549.976,A -85,B 0,C 180,E1 -32382.694,E2 -32382.694} C_VEL
LIN {X 0,Y 162.271,Z 552.135,A -85,B 0,C 180,E1 -32384.348,E2 -32384.348} C_VEL
LIN {X 0,Y 158.78,Z 556.111,A -85,B 0,C 180,E1 -32386.054,E2 -32386.054} C_VEL
LIN {X 0,Y 157.021,Z 557.91,A -85,B 0,C 180,E1 -32387.111,E2 -32387.111} C_VEL
LIN {X 0,Y 153.294,Z 561.362,A -85,B 0,C 180,E1 -32390.404,E2 -32390.404} C_VEL
LIN {X 0,Y 151.067,Z 563.973,A -85,B 0,C 180,E1 -32392.004,E2 -32392.004} C_VEL
LIN {X 0,Y 149.042,Z 566.062,A -85,B 0,C 180,E1 -32394.606,E2 -32394.606} C_VEL
LIN {X 0,Y 148.224,Z 566.972,A -85,B 0,C 180,E1 -32396.07,E2 -32396.07} C_VEL
LIN {X 0,Y 146.897,Z 568.794,A -85,B 0,C 180,E1 -32397.266,E2 -32397.266} C_VEL
LIN {X 0,Y 145.787,Z 570.4,A -85,B 0,C 180,E1 -32398.623,E2 -32398.623} C_VEL
LIN {X 0,Y 144.635,Z 572.688,A -85,B 0,C 180,E1 -32402.775,E2 -32402.775} C_VEL
LIN {X 0,Y 143.599,Z 574.543,A -85,B 0,C 180,E1 -32404.195,E2 -32404.195} C_VEL
LIN {X 0,Y 142.969,Z 575.97,A -85,B 0,C 180,E1 -32405.622,E2 -32405.622} C_VEL
LIN {X 0,Y 143.212,Z 577.156,A -85,B 0,C 180,E1 -32408.437,E2 -32408.437} C_VEL
LIN {X 0,Y 143.802,Z 576.748,A -85,B 0,C 180,E1 -32409.019,E2 -32409.019} C_VEL
LIN {X 0,Y 145.79,Z 587.605,A -85,B 0,C 180,E1 -32413.899,E2 -32413.899} C_VEL
LIN {X 0,Y 149.428,Z 597.867,A -85,B 0,C 180,E1 -32419.154,E2 -32419.154} C_VEL
LIN {X 0,Y 154.338,Z 606.608,A -85,B 0,C 180,E1 -32424.107,E2 -32424.107} C_VEL
LIN {X 0,Y 160.896,Z 614.056,A -85,B 0,C 180,E1 -32428.611,E2 -32428.611} C_VEL
LIN {X 0,Y 168.849,Z 620.317,A -85,B 0,C 180,E1 -32432.634,E2 -32432.634} C_VEL
LIN {X 0,Y 177.685,Z 625.366,A -85,B 0,C 180,E1 -32436.249,E2 -32436.249} C_VEL
LIN {X 0,Y 187.466,Z 629.288,A -85,B 0,C 180,E1 -32439.433,E2 -32439.433} C_VEL
LIN {X 0,Y 191.109,Z 630.44,A -85,B 0,C 180,E1 -32440.463,E2 -32440.463} C_VEL
LIN {X 0,Y 190.096,Z 630.788,A -85,B 0,C 180,E1 -32441.379,E2 -32441.379} C_VEL
LIN {X 0,Y 178.412,Z 630.202,A -85,B 0,C 180,E1 -32445.034,E2 -32445.034} C_VEL
LIN {X 0,Y 169.696,Z 628.896,A -85,B 0,C 180,E1 -32448.667,E2 -32448.667} C_VEL
LIN {X 0,Y 160.941,Z 626.494,A -85,B 0,C 180,E1 -32453.533,E2 -32453.533} C_VEL
LIN {X 0,Y 154.255,Z 632.94,A -85,B 0,C 180,E1 -32456.982,E2 -32456.982} C_VEL
LIN {X 0,Y 149.367,Z 637.755,A -85,B 0,C 180,E1 -32460.502,E2 -32460.502} C_VEL
LIN {X 0,Y 144.16,Z 642.825,A -85,B 0,C 180,E1 -32465.606,E2 -32465.606} C_VEL
LIN {X 0,Y 140.299,Z 646.708,A -85,B 0,C 180,E1 -32471.544,E2 -32471.544} C_VEL
LIN {X 0,Y 139.033,Z 648.311,A -85,B 0,C 180,E1 -32475.41,E2 -32475.41} C_VEL
LIN {X 0,Y 138.641,Z 649.675,A -85,B 0,C 180,E1 -32481.282,E2 -32481.282} C_VEL
LIN {X 0,Y 140.244,Z 649.784,A -85,B 0,C 180,E1 -32487.291,E2 -32487.291} C_VEL
LIN {X 0,Y 143.769,Z 648.702,A -85,B 0,C 180,E1 -32492.792,E2 -32492.792} C_VEL
LIN {X 0,Y 145.349,Z 648.123,A -85,B 0,C 180,E1 -32494.578,E2 -32494.578} C_VEL
LIN {X 0,Y 145.369,Z 655.187,A -85,B 0,C 180,E1 -32497.614,E2 -32497.614} C_VEL
LIN {X 0,Y 145.129,Z 663.376,A -85,B 0,C 180,E1 -32501.978,E2 -32501.978} C_VEL
LIN {X 0,Y 145.676,Z 670.842,A -85,B 0,C 180,E1 -32506.704,E2 -32506.704} C_VEL
LIN {X 0,Y 145.669,Z 673.475,A -85,B 0,C 180,E1 -32508.788,E2 -32508.788} C_VEL
LIN {X 0,Y 144.785,Z 676.774,A -85,B 0,C 180,E1 -32512.468,E2 -32512.468} C_VEL
LIN {X 0,Y 144.776,Z 679.866,A -85,B 0,C 180,E1 -32516.197,E2 -32516.197} C_VEL
LIN {X 0,Y 146.063,Z 682.115,A -85,B 0,C 180,E1 -32518.282,E2 -32518.282} C_VEL
LIN {X 0,Y 152.175,Z 688.373,A -85,B 0,C 180,E1 -32523.528,E2 -32523.528} C_VEL
LIN {X 0,Y 161.315,Z 694.341,A -85,B 0,C 180,E1 -32529.02,E2 -32529.02} C_VEL
LIN {X 0,Y 167.807,Z 697.324,A -85,B 0,C 180,E1 -32531.901,E2 -32531.901} C_VEL
LIN {X 0,Y 175.735,Z 700.006,A -85,B 0,C 180,E1 -32534.749,E2 -32534.749} C_VEL
LIN {X 0,Y 174.817,Z 699.727,A -85,B 0,C 180,E1 -32535.773,E2 -32535.773} C_VEL
LIN {X 0,Y 163.698,Z 695.426,A -85,B 0,C 180,E1 -32540.072,E2 -32540.072} C_VEL
LIN {X 0,Y 154.259,Z 689.822,A -85,B 0,C 180,E1 -32545.228,E2 -32545.228} C_VEL
LIN {X 0,Y 146.446,Z 682.388,A -85,B 0,C 180,E1 -32551.427,E2 -32551.427} C_VEL
LIN {X 0,Y 142.168,Z 675.437,A -85,B 0,C 180,E1 -32556.788,E2 -32556.788} C_VEL
LIN {X 0,Y 139.464,Z 666.167,A -85,B 0,C 180,E1 -32563.211,E2 -32563.211} C_VEL
LIN {X 0,Y 138.891,Z 657.727,A -85,B 0,C 180,E1 -32568.363,E2 -32568.363} C_VEL
LIN {X 0,Y 139.093,Z 649.112,A -85,B 0,C 180,E1 -32572.768,E2 -32572.768} C_VEL
LIN {X 0,Y 138.881,Z 641.927,A -85,B 0,C 180,E1 -32575.662,E2 -32575.662} C_VEL
LIN {X 0,Y 138.47,Z 631.13,A -85,B 0,C 180,E1 -32579.276,E2 -32579.276} C_VEL
LIN {X 0,Y 138.243,Z 619.345,A -85,B 0,C 180,E1 -32582.542,E2 -32582.542} C_VEL
LIN {X 0,Y 138.121,Z 604.589,A -85,B 0,C 180,E1 -32585.822,E2 -32585.822} C_VEL
LIN {X 0,Y 138.272,Z 590.128,A -85,B 0,C 180,E1 -32588.375,E2 -32588.375} C_VEL
LIN {X 0,Y 138.36,Z 574.948,A -85,B 0,C 180,E1 -32590.391,E2 -32590.391} C_VEL
LIN {X 0,Y 138.443,Z 534.987,A -85,B 0,C 180,E1 -32594.845,E2 -32594.845} C_VEL
LIN {X 0,Y 139.512,Z 481.041,A -85,B 0,C 180,E1 -32600.673,E2 -32600.673} C_VEL
LIN {X 0,Y 138.298,Z 466.629,A -85,B 0,C 180,E1 -32602.13,E2 -32602.13} C_VEL
LIN {X 0,Y 138.396,Z 468.908,A -85,B 0,C 180,E1 -32602.603,E2 -32602.603} C_VEL
LIN {X 0,Y 138.681,Z 469.614,A -85,B 0,C 180,E1 -32603.045,E2 -32603.045} C_VEL
LIN {X 0,Y 139.321,Z 469.261,A -85,B 0,C 180,E1 -32603.717,E2 -32603.717} C_VEL
LIN {X 0,Y 140.516,Z 466.715,A -85,B 0,C 180,E1 -32604.643,E2 -32604.643} C_VEL
LIN {X 0,Y 142.314,Z 461.065,A -85,B 0,C 180,E1 -32605.706,E2 -32605.706} C_VEL
LIN {X 0,Y 145.016,Z 450.536,A -85,B 0,C 180,E1 -32606.926,E2 -32606.926} C_VEL
LIN {X 0,Y 146.633,Z 448.88,A -85,B 0,C 180,E1 -32608.146,E2 -32608.146} C_VEL
LIN {X 0,Y 148.31,Z 446.384,A -85,B 0,C 180,E1 -32609.244,E2 -32609.244} C_VEL
LIN {X 0,Y 151.725,Z 441.322,A -85,B 0,C 180,E1 -32611.29,E2 -32611.29} C_VEL
LIN {X 0,Y 153.725,Z 437.914,A -85,B 0,C 180,E1 -32612.347,E2 -32612.347} C_VEL
LIN {X 0,Y 156.915,Z 436.329,A -85,B 0,C 180,E1 -32614.248,E2 -32614.248} C_VEL
LIN {X 0,Y 160.591,Z 432.803,A -85,B 0,C 180,E1 -32616.093,E2 -32616.093} C_VEL
LIN {X 0,Y 161.952,Z 431.499,A -85,B 0,C 180,E1 -32616.733,E2 -32616.733} C_VEL
LIN {X 0,Y 165.719,Z 430.102,A -85,B 0,C 180,E1 -32618.562,E2 -32618.562} C_VEL
LIN {X 0,Y 168.089,Z 429.495,A -85,B 0,C 180,E1 -32619.65,E2 -32619.65} C_VEL
LIN {X 0,Y 169.604,Z 429.627,A -85,B 0,C 180,E1 -32620.352,E2 -32620.352} C_VEL
LIN {X 0,Y 175.441,Z 440.73,A -85,B 0,C 180,E1 -32623.515,E2 -32623.515} C_VEL
LIN {X 0,Y 178.906,Z 448.44,A -85,B 0,C 180,E1 -32625.273,E2 -32625.273} C_VEL
LIN {X 0,Y 175.88,Z 496.165,A -85,B 0,C 180,E1 -32627.082,E2 -32627.082} C_VEL
LIN {X 0,Y 174.183,Z 510.781,A -85,B 0,C 180,E1 -32628.045,E2 -32628.045} C_VEL
LIN {X 0,Y 171.826,Z 524.019,A -85,B 0,C 180,E1 -32629.29,E2 -32629.29} C_VEL
LIN {X 0,Y 168.838,Z 536.138,A -85,B 0,C 180,E1 -32630.753,E2 -32630.753} C_VEL
LIN {X 0,Y 165.559,Z 547.423,A -85,B 0,C 180,E1 -32632.543,E2 -32632.543} C_VEL
LIN {X 0,Y 161.494,Z 559.196,A -85,B 0,C 180,E1 -32634.922,E2 -32634.922} C_VEL
LIN {X 0,Y 157.052,Z 569.976,A -85,B 0,C 180,E1 -32637.643,E2 -32637.643} C_VEL
LIN {X 0,Y 152.637,Z 579.42,A -85,B 0,C 180,E1 -32640.626,E2 -32640.626} C_VEL
LIN {X 0,Y 148.008,Z 588.571,A -85,B 0,C 180,E1 -32644.309,E2 -32644.309} C_VEL
LIN {X 0,Y 143.706,Z 596.738,A -85,B 0,C 180,E1 -32648.558,E2 -32648.558} C_VEL
LIN {X 0,Y 140.199,Z 602.877,A -85,B 0,C 180,E1 -32652.557,E2 -32652.557} C_VEL
LIN {X 0,Y 136.616,Z 609.375,A -85,B 0,C 180,E1 -32658.166,E2 -32658.166} C_VEL
LIN {X 0,Y 134.131,Z 614.271,A -85,B 0,C 180,E1 -32664.005,E2 -32664.005} C_VEL
LIN {X 0,Y 132.912,Z 617.704,A -85,B 0,C 180,E1 -32670,E2 -32670} C_VEL
LIN {X 0,Y 132.797,Z 619.797,A -85,B 0,C 180,E1 -32676.056,E2 -32676.056} C_VEL
LIN {X 0,Y 133.726,Z 620.606,A -85,B 0,C 180,E1 -32682.095,E2 -32682.095} C_VEL
LIN {X 0,Y 135.767,Z 620.129,A -85,B 0,C 180,E1 -32688.033,E2 -32688.033} C_VEL
LIN {X 0,Y 139.201,Z 618.309,A -85,B 0,C 180,E1 -32693.738,E2 -32693.738} C_VEL
LIN {X 0,Y 143.707,Z 615.112,A -85,B 0,C 180,E1 -32699.171,E2 -32699.171} C_VEL
LIN {X 0,Y 149.216,Z 610.441,A -85,B 0,C 180,E1 -32704.285,E2 -32704.285} C_VEL
LIN {X 0,Y 155.673,Z 604.145,A -85,B 0,C 180,E1 -32709.045,E2 -32709.045} C_VEL
LIN {X 0,Y 161.403,Z 597.809,A -85,B 0,C 180,E1 -32712.569,E2 -32712.569} C_VEL
LIN {X 0,Y 167.993,Z 589.676,A -85,B 0,C 180,E1 -32715.992,E2 -32715.992} C_VEL
LIN {X 0,Y 174.408,Z 580.727,A -85,B 0,C 180,E1 -32718.854,E2 -32718.854} C_VEL
LIN {X 0,Y 180.526,Z 570.56,A -85,B 0,C 180,E1 -32721.47,E2 -32721.47} C_VEL
LIN {X 0,Y 186.13,Z 559.948,A -85,B 0,C 180,E1 -32723.552,E2 -32723.552} C_VEL
LIN {X 0,Y 191.54,Z 547.946,A -85,B 0,C 180,E1 -32725.367,E2 -32725.367} C_VEL
LIN {X 0,Y 195.676,Z 536.359,A -85,B 0,C 180,E1 -32726.798,E2 -32726.798} C_VEL
LIN {X 0,Y 199.471,Z 522.73,A -85,B 0,C 180,E1 -32728.108,E2 -32728.108} C_VEL
LIN {X 0,Y 202.242,Z 508.884,A -85,B 0,C 180,E1 -32729.096,E2 -32729.096} C_VEL
LIN {X 0,Y 203.555,Z 499.575,A -85,B 0,C 180,E1 -32729.582,E2 -32729.582} C_VEL
LIN {X 0,Y 199.357,Z 506.859,A -85,B 0,C 180,E1 -32730.72,E2 -32730.72} C_VEL
LIN {X 0,Y 197.373,Z 509.98,A -85,B 0,C 180,E1 -32731.276,E2 -32731.276} C_VEL
LIN {X 0,Y 192.907,Z 519.349,A -85,B 0,C 180,E1 -32732.022,E2 -32732.022} C_VEL
LIN {X 0,Y 188.371,Z 526.926,A -85,B 0,C 180,E1 -32732.902,E2 -32732.902} C_VEL
LIN {X 0,Y 183.55,Z 533.516,A -85,B 0,C 180,E1 -32734.065,E2 -32734.065} C_VEL
LIN {X 0,Y 178.338,Z 539.432,A -85,B 0,C 180,E1 -32735.644,E2 -32735.644} C_VEL
LIN {X 0,Y 174.725,Z 543.005,A -85,B 0,C 180,E1 -32736.928,E2 -32736.928} C_VEL
LIN {X 0,Y 170.154,Z 548.375,A -85,B 0,C 180,E1 -32738.254,E2 -32738.254} C_VEL
LIN {X 0,Y 165.207,Z 553.313,A -85,B 0,C 180,E1 -32740.172,E2 -32740.172} C_VEL
LIN {X 0,Y 162.555,Z 555.633,A -85,B 0,C 180,E1 -32741.438,E2 -32741.438} C_VEL
LIN {X 0,Y 160.144,Z 557.571,A -85,B 0,C 180,E1 -32742.828,E2 -32742.828} C_VEL
LIN {X 0,Y 155.666,Z 562.072,A -85,B 0,C 180,E1 -32744.953,E2 -32744.953} C_VEL
LIN {X 0,Y 152.934,Z 564.451,A -85,B 0,C 180,E1 -32746.761,E2 -32746.761} C_VEL
LIN {X 0,Y 149.941,Z 567.062,A -85,B 0,C 180,E1 -32749.23,E2 -32749.23} C_VEL
LIN {X 0,Y 148.275,Z 568.82,A -85,B 0,C 180,E1 -32750.345,E2 -32750.345} C_VEL
LIN {X 0,Y 146.779,Z 570.225,A -85,B 0,C 180,E1 -32751.768,E2 -32751.768} C_VEL
LIN {X 0,Y 144.823,Z 572.068,A -85,B 0,C 180,E1 -32754.448,E2 -32754.448} C_VEL
LIN {X 0,Y 142.158,Z 575.302,A -85,B 0,C 180,E1 -32757.175,E2 -32757.175} C_VEL
LIN {X 0,Y 140.181,Z 578.336,A -85,B 0,C 180,E1 -32762.06,E2 -32762.06} C_VEL
LIN {X 0,Y 138.756,Z 580.754,A -85,B 0,C 180,E1 -32764.342,E2 -32764.342} C_VEL
LIN {X 0,Y 138.511,Z 581.627,A -85,B 0,C 180,E1 -32765.804,E2 -32765.804} C_VEL
LIN {X 0,Y 138.846,Z 582.69,A -85,B 0,C 180,E1 -32768.704,E2 -32768.704} C_VEL
LIN {X 0,Y 138.106,Z 585.493,A -85,B 0,C 180,E1 -32771.704,E2 -32771.704} C_VEL
LIN {X 0,Y 138.971,Z 586.747,A -85,B 0,C 180,E1 -32774.596,E2 -32774.596} C_VEL
LIN {X 0,Y 140.026,Z 586.563,A -85,B 0,C 180,E1 -32775.596,E2 -32775.596} C_VEL
LIN {X 0,Y 144.202,Z 597.765,A -85,B 0,C 180,E1 -32781.364,E2 -32781.364} C_VEL
LIN {X 0,Y 149.666,Z 606.582,A -85,B 0,C 180,E1 -32786.397,E2 -32786.397} C_VEL
LIN {X 0,Y 156.726,Z 614.205,A -85,B 0,C 180,E1 -32790.927,E2 -32790.927} C_VEL
LIN {X 0,Y 165.145,Z 620.612,A -85,B 0,C 180,E1 -32794.93,E2 -32794.93} C_VEL
LIN {X 0,Y 174.446,Z 625.842,A -85,B 0,C 180,E1 -32798.488,E2 -32798.488} C_VEL
LIN {X 0,Y 180.723,Z 628.52,A -85,B 0,C 180,E1 -32800.48,E2 -32800.48} C_VEL
LIN {X 0,Y 179.166,Z 628.791,A -85,B 0,C 180,E1 -32801.652,E2 -32801.652} C_VEL
LIN {X 0,Y 169.039,Z 627.409,A -85,B 0,C 180,E1 -32805.216,E2 -32805.216} C_VEL
LIN {X 0,Y 158.751,Z 624.814,A -85,B 0,C 180,E1 -32810.224,E2 -32810.224} C_VEL
LIN {X 0,Y 156.861,Z 624.383,A -85,B 0,C 180,E1 -32811.306,E2 -32811.306} C_VEL
LIN {X 0,Y 150.349,Z 630.505,A -85,B 0,C 180,E1 -32814.383,E2 -32814.383} C_VEL
LIN {X 0,Y 144.84,Z 635.639,A -85,B 0,C 180,E1 -32817.861,E2 -32817.861} C_VEL
LIN {X 0,Y 138.934,Z 641.032,A -85,B 0,C 180,E1 -32823.016,E2 -32823.016} C_VEL
LIN {X 0,Y 134.649,Z 644.969,A -85,B 0,C 180,E1 -32828.645,E2 -32828.645} C_VEL
LIN {X 0,Y 132.114,Z 647.566,A -85,B 0,C 180,E1 -32834.627,E2 -32834.627} C_VEL
LIN {X 0,Y 131.558,Z 648.902,A -85,B 0,C 180,E1 -32840.808,E2 -32840.808} C_VEL
LIN {X 0,Y 133.202,Z 648.937,A -85,B 0,C 180,E1 -32847.583,E2 -32847.583} C_VEL
LIN {X 0,Y 136.525,Z 647.865,A -85,B 0,C 180,E1 -32852.94,E2 -32852.94} C_VEL
LIN {X 0,Y 139.308,Z 646.843,A -85,B 0,C 180,E1 -32856.133,E2 -32856.133} C_VEL
LIN {X 0,Y 139.275,Z 653.982,A -85,B 0,C 180,E1 -32859.407,E2 -32859.407} C_VEL
LIN {X 0,Y 139.291,Z 663.035,A -85,B 0,C 180,E1 -32864.562,E2 -32864.562} C_VEL
LIN {X 0,Y 140.729,Z 671.729,A -85,B 0,C 180,E1 -32870.39,E2 -32870.39} C_VEL
LIN {X 0,Y 143.969,Z 679.143,A -85,B 0,C 180,E1 -32875.968,E2 -32875.968} C_VEL
LIN {X 0,Y 146.063,Z 682.115,A -85,B 0,C 180,E1 -32878.282,E2 -32878.282} C_VEL
LIN {X 0,Y 147.58,Z 684.327,A -85,B 0,C 180,E1 -32880.334,E2 -32880.334} C_VEL
LIN {X 0,Y 149.138,Z 686.967,A -85,B 0,C 180,E1 -32883.976,E2 -32883.976} C_VEL
LIN {X 0,Y 150.794,Z 688.773,A -85,B 0,C 180,E1 -32886.873,E2 -32886.873} C_VEL
LIN {X 0,Y 152.961,Z 690.329,A -85,B 0,C 180,E1 -32888.872,E2 -32888.872} C_VEL
LIN {X 0,Y 153.935,Z 690.924,A -85,B 0,C 180,E1 -32889.473,E2 -32889.473} C_VEL
LIN {X 0,Y 162.789,Z 695.429,A -85,B 0,C 180,E1 -32893.507,E2 -32893.507} C_VEL
LIN {X 0,Y 166.037,Z 696.736,A -85,B 0,C 180,E1 -32894.736,E2 -32894.736} C_VEL
LIN {X 0,Y 165.099,Z 696.347,A -85,B 0,C 180,E1 -32895.835,E2 -32895.835} C_VEL
LIN {X 0,Y 154.303,Z 691.038,A -85,B 0,C 180,E1 -32900.542,E2 -32900.542} C_VEL
LIN {X 0,Y 145.241,Z 684.282,A -85,B 0,C 180,E1 -32906.317,E2 -32906.317} C_VEL
LIN {X 0,Y 138.306,Z 675.937,A -85,B 0,C 180,E1 -32912.884,E2 -32912.884} C_VEL
LIN {X 0,Y 134.411,Z 666.538,A -85,B 0,C 180,E1 -32919.721,E2 -32919.721} C_VEL
LIN {X 0,Y 133.171,Z 657.647,A -85,B 0,C 180,E1 -32925.533,E2 -32925.533} C_VEL
LIN {X 0,Y 133.145,Z 647.848,A -85,B 0,C 180,E1 -32930.92,E2 -32930.92} C_VEL
LIN {X 0,Y 132.946,Z 640.788,A -85,B 0,C 180,E1 -32933.952,E2 -32933.952} C_VEL
LIN {X 0,Y 132.379,Z 630.019,A -85,B 0,C 180,E1 -32937.726,E2 -32937.726} C_VEL
LIN {X 0,Y 132.03,Z 618.195,A -85,B 0,C 180,E1 -32941.141,E2 -32941.141} C_VEL
LIN {X 0,Y 131.754,Z 603.458,A -85,B 0,C 180,E1 -32944.575,E2 -32944.575} C_VEL
LIN {X 0,Y 131.848,Z 590.021,A -85,B 0,C 180,E1 -32947.058,E2 -32947.058} C_VEL
LIN {X 0,Y 131.86,Z 574.979,A -85,B 0,C 180,E1 -32949.171,E2 -32949.171} C_VEL
LIN {X 0,Y 131.674,Z 531.312,A -85,B 0,C 180,E1 -32954.342,E2 -32954.342} C_VEL
LIN {X 0,Y 132.22,Z 494.307,A -85,B 0,C 180,E1 -32958.584,E2 -32958.584} C_VEL
LIN {X 0,Y 131.976,Z 497.857,A -85,B 0,C 180,E1 -32958.971,E2 -32958.971} C_VEL
LIN {X 0,Y 132.073,Z 499.036,A -85,B 0,C 180,E1 -32959.359,E2 -32959.359} C_VEL
LIN {X 0,Y 132.461,Z 498.869,A -85,B 0,C 180,E1 -32959.903,E2 -32959.903} C_VEL
LIN {X 0,Y 133.329,Z 496.928,A -85,B 0,C 180,E1 -32960.771,E2 -32960.771} C_VEL
LIN {X 0,Y 135.061,Z 491.117,A -85,B 0,C 180,E1 -32962.057,E2 -32962.057} C_VEL
LIN {X 0,Y 138.291,Z 478.402,A -85,B 0,C 180,E1 -32963.905,E2 -32963.905} C_VEL
LIN {X 0,Y 138.767,Z 476.446,A -85,B 0,C 180,E1 -32964.144,E2 -32964.144} C_VEL
LIN {X 0,Y 140.261,Z 474.872,A -85,B 0,C 180,E1 -32965.489,E2 -32965.489} C_VEL
LIN {X 0,Y 142.028,Z 471.354,A -85,B 0,C 180,E1 -32966.746,E2 -32966.746} C_VEL
LIN {X 0,Y 144.133,Z 465.403,A -85,B 0,C 180,E1 -32967.92,E2 -32967.92} C_VEL
LIN {X 0,Y 146.866,Z 455.742,A -85,B 0,C 180,E1 -32969.111,E2 -32969.111} C_VEL
LIN {X 0,Y 152.449,Z 448.082,A -85,B 0,C 180,E1 -32972.45,E2 -32972.45} C_VEL
LIN {X 0,Y 154.988,Z 444.352,A -85,B 0,C 180,E1 -32973.763,E2 -32973.763} C_VEL
LIN {X 0,Y 158.706,Z 442.03,A -85,B 0,C 180,E1 -32975.789,E2 -32975.789} C_VEL
LIN {X 0,Y 162.628,Z 438.293,A -85,B 0,C 180,E1 -32977.62,E2 -32977.62} C_VEL
LIN {X 0,Y 166.094,Z 436.912,A -85,B 0,C 180,E1 -32979.241,E2 -32979.241} C_VEL
LIN {X 0,Y 167.453,Z 437.154,A -85,B 0,C 180,E1 -32979.898,E2 -32979.898} C_VEL
LIN {X 0,Y 172.264,Z 446.762,A -85,B 0,C 180,E1 -32982.635,E2 -32982.635} C_VEL
LIN {X 0,Y 174.013,Z 450.653,A -85,B 0,C 180,E1 -32983.58,E2 -32983.58} C_VEL
LIN {X 0,Y 170.995,Z 497.308,A -85,B 0,C 180,E1 -32985.419,E2 -32985.419} C_VEL
LIN {X 0,Y 169.173,Z 511.923,A -85,B 0,C 180,E1 -32986.399,E2 -32986.399} C_VEL
LIN {X 0,Y 166.541,Z 525.631,A -85,B 0,C 180,E1 -32987.706,E2 -32987.706} C_VEL
LIN {X 0,Y 162.957,Z 539.293,A -85,B 0,C 180,E1 -32989.449,E2 -32989.449} C_VEL
LIN {X 0,Y 159.091,Z 551.512,A -85,B 0,C 180,E1 -32991.546,E2 -32991.546} C_VEL
LIN {X 0,Y 154.862,Z 562.702,A -85,B 0,C 180,E1 -32993.986,E2 -32993.986} C_VEL
LIN {X 0,Y 150.249,Z 573.025,A -85,B 0,C 180,E1 -32996.786,E2 -32996.786} C_VEL
LIN {X 0,Y 145.003,Z 583.462,A -85,B 0,C 180,E1 -33000.402,E2 -33000.402} C_VEL
LIN {X 0,Y 139.839,Z 593.027,A -85,B 0,C 180,E1 -33004.802,E2 -33004.802} C_VEL
LIN {X 0,Y 135.869,Z 599.902,A -85,B 0,C 180,E1 -33008.847,E2 -33008.847} C_VEL
LIN {X 0,Y 132.454,Z 605.59,A -85,B 0,C 180,E1 -33013.091,E2 -33013.091} C_VEL
LIN {X 0,Y 129.721,Z 610.273,A -85,B 0,C 180,E1 -33017.527,E2 -33017.527} C_VEL
LIN {X 0,Y 127.112,Z 615.137,A -85,B 0,C 180,E1 -33023.673,E2 -33023.673} C_VEL
LIN {X 0,Y 125.857,Z 618.538,A -85,B 0,C 180,E1 -33030.001,E2 -33030.001} C_VEL
LIN {X 0,Y 125.771,Z 620.602,A -85,B 0,C 180,E1 -33036.396,E2 -33036.396} C_VEL
LIN {X 0,Y 126.815,Z 621.382,A -85,B 0,C 180,E1 -33042.764,E2 -33042.764} C_VEL
LIN {X 0,Y 129.031,Z 620.872,A -85,B 0,C 180,E1 -33049.009,E2 -33049.009} C_VEL
LIN {X 0,Y 132.74,Z 619.013,A -85,B 0,C 180,E1 -33054.971,E2 -33054.971} C_VEL
LIN {X 0,Y 137.548,Z 615.784,A -85,B 0,C 180,E1 -33060.614,E2 -33060.614} C_VEL
LIN {X 0,Y 143.398,Z 611.08,A -85,B 0,C 180,E1 -33065.885,E2 -33065.885} C_VEL
LIN {X 0,Y 150.223,Z 604.748,A -85,B 0,C 180,E1 -33070.752,E2 -33070.752} C_VEL
LIN {X 0,Y 156.982,Z 597.558,A -85,B 0,C 180,E1 -33074.735,E2 -33074.735} C_VEL
LIN {X 0,Y 164.211,Z 588.841,A -85,B 0,C 180,E1 -33078.286,E2 -33078.286} C_VEL
LIN {X 0,Y 170.937,Z 579.534,A -85,B 0,C 180,E1 -33081.129,E2 -33081.129} C_VEL
LIN {X 0,Y 177.009,Z 569.531,A -85,B 0,C 180,E1 -33083.589,E2 -33083.589} C_VEL
LIN {X 0,Y 182.622,Z 559.041,A -85,B 0,C 180,E1 -33085.552,E2 -33085.552} C_VEL
LIN {X 0,Y 188.216,Z 546.577,A -85,B 0,C 180,E1 -33087.352,E2 -33087.352} C_VEL
LIN {X 0,Y 192.484,Z 534.466,A -85,B 0,C 180,E1 -33088.778,E2 -33088.778} C_VEL
LIN {X 0,Y 196.06,Z 521.303,A -85,B 0,C 180,E1 -33089.988,E2 -33089.988} C_VEL
LIN {X 0,Y 194.711,Z 523.089,A -85,B 0,C 180,E1 -33090.314,E2 -33090.314} C_VEL
LIN {X 0,Y 189.282,Z 531.473,A -85,B 0,C 180,E1 -33091.244,E2 -33091.244} C_VEL
LIN {X 0,Y 184.014,Z 538.074,A -85,B 0,C 180,E1 -33092.378,E2 -33092.378} C_VEL
LIN {X 0,Y 178.744,Z 543.614,A -85,B 0,C 180,E1 -33093.784,E2 -33093.784} C_VEL
LIN {X 0,Y 174.653,Z 547.424,A -85,B 0,C 180,E1 -33095.095,E2 -33095.095} C_VEL
LIN {X 0,Y 169.974,Z 552.52,A -85,B 0,C 180,E1 -33096.31,E2 -33096.31} C_VEL
LIN {X 0,Y 164.586,Z 557.493,A -85,B 0,C 180,E1 -33098.137,E2 -33098.137} C_VEL
LIN {X 0,Y 161.051,Z 560.438,A -85,B 0,C 180,E1 -33099.638,E2 -33099.638} C_VEL
LIN {X 0,Y 158.596,Z 562.198,A -85,B 0,C 180,E1 -33100.957,E2 -33100.957} C_VEL
LIN {X 0,Y 153.774,Z 566.619,A -85,B 0,C 180,E1 -33103.052,E2 -33103.052} C_VEL
LIN {X 0,Y 152.033,Z 568.077,A -85,B 0,C 180,E1 -33103.952,E2 -33103.952} C_VEL
LIN {X 0,Y 146.998,Z 571.977,A -85,B 0,C 180,E1 -33107.617,E2 -33107.617} C_VEL
LIN {X 0,Y 145.022,Z 573.849,A -85,B 0,C 180,E1 -33108.86,E2 -33108.86} C_VEL
LIN {X 0,Y 142.312,Z 576.108,A -85,B 0,C 180,E1 -33111.508,E2 -33111.508} C_VEL
LIN {X 0,Y 141.129,Z 577.127,A -85,B 0,C 180,E1 -33113.045,E2 -33113.045} C_VEL
LIN {X 0,Y 138.417,Z 580.013,A -85,B 0,C 180,E1 -33115.646,E2 -33115.646} C_VEL
LIN {X 0,Y 135.731,Z 583.427,A -85,B 0,C 180,E1 -33121.009,E2 -33121.009} C_VEL
LIN {X 0,Y 134.416,Z 585.349,A -85,B 0,C 180,E1 -33122.986,E2 -33122.986} C_VEL
LIN {X 0,Y 133.602,Z 588.746,A -85,B 0,C 180,E1 -33129.048,E2 -33129.048} C_VEL
LIN {X 0,Y 133.242,Z 590.014,A -85,B 0,C 180,E1 -33130.602,E2 -33130.602} C_VEL
LIN {X 0,Y 133.352,Z 590.842,A -85,B 0,C 180,E1 -33132.128,E2 -33132.128} C_VEL
LIN {X 0,Y 134.339,Z 591.985,A -85,B 0,C 180,E1 -33135.111,E2 -33135.111} C_VEL
LIN {X 0,Y 134.923,Z 593.944,A -85,B 0,C 180,E1 -33138.148,E2 -33138.148} C_VEL
LIN {X 0,Y 136.453,Z 595.28,A -85,B 0,C 180,E1 -33141.058,E2 -33141.058} C_VEL
LIN {X 0,Y 138.259,Z 595.423,A -85,B 0,C 180,E1 -33142.625,E2 -33142.625} C_VEL
LIN {X 0,Y 144.4,Z 605.392,A -85,B 0,C 180,E1 -33148.225,E2 -33148.225} C_VEL
LIN {X 0,Y 152.836,Z 614.206,A -85,B 0,C 180,E1 -33153.363,E2 -33153.363} C_VEL
LIN {X 0,Y 161.719,Z 620.807,A -85,B 0,C 180,E1 -33157.327,E2 -33157.327} C_VEL
LIN {X 0,Y 171.477,Z 626.203,A -85,B 0,C 180,E1 -33160.81,E2 -33160.81} C_VEL
LIN {X 0,Y 169.121,Z 625.937,A -85,B 0,C 180,E1 -33161.797,E2 -33161.797} C_VEL
LIN {X 0,Y 159.936,Z 623.989,A -85,B 0,C 180,E1 -33165.514,E2 -33165.514} C_VEL
LIN {X 0,Y 153.407,Z 622.001,A -85,B 0,C 180,E1 -33168.869,E2 -33168.869} C_VEL
LIN {X 0,Y 146.765,Z 627.984,A -85,B 0,C 180,E1 -33171.652,E2 -33171.652} C_VEL
LIN {X 0,Y 140.69,Z 633.374,A -85,B 0,C 180,E1 -33175.071,E2 -33175.071} C_VEL
LIN {X 0,Y 134.066,Z 639.144,A -85,B 0,C 180,E1 -33180.241,E2 -33180.241} C_VEL
LIN {X 0,Y 130.152,Z 642.48,A -85,B 0,C 180,E1 -33184.498,E2 -33184.498} C_VEL
LIN {X 0,Y 126.357,Z 645.697,A -85,B 0,C 180,E1 -33190.573,E2 -33190.573} C_VEL
LIN {X 0,Y 124.6,Z 647.631,A -85,B 0,C 180,E1 -33197.005,E2 -33197.005} C_VEL
LIN {X 0,Y 124.887,Z 648.316,A -85,B 0,C 180,E1 -33203.559,E2 -33203.559} C_VEL
LIN {X 0,Y 127.233,Z 647.759,A -85,B 0,C 180,E1 -33210,E2 -33210} C_VEL
LIN {X 0,Y 131.75,Z 645.971,A -85,B 0,C 180,E1 -33216.103,E2 -33216.103} C_VEL
LIN {X 0,Y 133.383,Z 645.406,A -85,B 0,C 180,E1 -33217.828,E2 -33217.828} C_VEL
LIN {X 0,Y 133.38,Z 651.181,A -85,B 0,C 180,E1 -33220.591,E2 -33220.591} C_VEL
LIN {X 0,Y 133.555,Z 660.639,A -85,B 0,C 180,E1 -33226.139,E2 -33226.139} C_VEL
LIN {X 0,Y 135.565,Z 670.299,A -85,B 0,C 180,E1 -33232.799,E2 -33232.799} C_VEL
LIN {X 0,Y 139.41,Z 677.809,A -85,B 0,C 180,E1 -33238.51,E2 -33238.51} C_VEL
LIN {X 0,Y 145.065,Z 684.315,A -85,B 0,C 180,E1 -33243.729,E2 -33243.729} C_VEL
LIN {X 0,Y 153.935,Z 690.924,A -85,B 0,C 180,E1 -33249.473,E2 -33249.473} C_VEL
LIN {X 0,Y 155.136,Z 691.678,A -85,B 0,C 180,E1 -33250.38,E2 -33250.38} C_VEL
LIN {X 0,Y 156.013,Z 692.305,A -85,B 0,C 180,E1 -33251.902,E2 -33251.902} C_VEL
LIN {X 0,Y 156.026,Z 692.408,A -85,B 0,C 180,E1 -33253.488,E2 -33253.488} C_VEL
LIN {X 0,Y 155.298,Z 692.079,A -85,B 0,C 180,E1 -33255.07,E2 -33255.07} C_VEL
LIN {X 0,Y 153.803,Z 691.262,A -85,B 0,C 180,E1 -33256.551,E2 -33256.551} C_VEL
LIN {X 0,Y 152.296,Z 690.436,A -85,B 0,C 180,E1 -33257.417,E2 -33257.417} C_VEL
LIN {X 0,Y 143.389,Z 684.483,A -85,B 0,C 180,E1 -33262.367,E2 -33262.367} C_VEL
LIN {X 0,Y 135.276,Z 676.343,A -85,B 0,C 180,E1 -33268.817,E2 -33268.817} C_VEL
LIN {X 0,Y 130.092,Z 667.15,A -85,B 0,C 180,E1 -33275.718,E2 -33275.718} C_VEL
LIN {X 0,Y 127.837,Z 658.377,A -85,B 0,C 180,E1 -33281.781,E2 -33281.781} C_VEL
LIN {X 0,Y 127.289,Z 649.357,A -85,B 0,C 180,E1 -33287.285,E2 -33287.285} C_VEL
LIN {X 0,Y 127.31,Z 643.191,A -85,B 0,C 180,E1 -33290.5,E2 -33290.5} C_VEL
LIN {X 0,Y 126.883,Z 635.513,A -85,B 0,C 180,E1 -33293.662,E2 -33293.662} C_VEL
LIN {X 0,Y 126.189,Z 623.796,A -85,B 0,C 180,E1 -33297.613,E2 -33297.613} C_VEL
LIN {X 0,Y 125.782,Z 612.403,A -85,B 0,C 180,E1 -33300.799,E2 -33300.799} C_VEL
LIN {X 0,Y 125.515,Z 598.208,A -85,B 0,C 180,E1 -33304.001,E2 -33304.001} C_VEL
LIN {X 0,Y 125.468,Z 584.078,A -85,B 0,C 180,E1 -33306.512,E2 -33306.512} C_VEL
LIN {X 0,Y 125.292,Z 561.288,A -85,B 0,C 180,E1 -33309.554,E2 -33309.554} C_VEL
LIN {X 0,Y 124.901,Z 521.525,A -85,B 0,C 180,E1 -33314.462,E2 -33314.462} C_VEL
LIN {X 0,Y 124.589,Z 523.534,A -85,B 0,C 180,E1 -33315.176,E2 -33315.176} C_VEL
LIN {X 0,Y 124.634,Z 523.82,A -85,B 0,C 180,E1 -33315.484,E2 -33315.484} C_VEL
LIN {X 0,Y 125.154,Z 523.635,A -85,B 0,C 180,E1 -33316.522,E2 -33316.522} C_VEL
LIN {X 0,Y 126.32,Z 521.456,A -85,B 0,C 180,E1 -33317.583,E2 -33317.583} C_VEL
LIN {X 0,Y 128.473,Z 516.248,A -85,B 0,C 180,E1 -33318.927,E2 -33318.927} C_VEL
LIN {X 0,Y 131.16,Z 507.907,A -85,B 0,C 180,E1 -33320.21,E2 -33320.21} C_VEL
LIN {X 0,Y 131.685,Z 506.041,A -85,B 0,C 180,E1 -33320.431,E2 -33320.431} C_VEL
LIN {X 0,Y 133.088,Z 504.357,A -85,B 0,C 180,E1 -33321.923,E2 -33321.923} C_VEL
LIN {X 0,Y 134.747,Z 500.687,A -85,B 0,C 180,E1 -33323.272,E2 -33323.272} C_VEL
LIN {X 0,Y 136.573,Z 495.235,A -85,B 0,C 180,E1 -33324.448,E2 -33324.448} C_VEL
LIN {X 0,Y 140.122,Z 482.334,A -85,B 0,C 180,E1 -33326.329,E2 -33326.329} C_VEL
LIN {X 0,Y 140.434,Z 481.622,A -85,B 0,C 180,E1 -33326.538,E2 -33326.538} C_VEL
LIN {X 0,Y 142.448,Z 478.587,A -85,B 0,C 180,E1 -33328.005,E2 -33328.005} C_VEL
LIN {X 0,Y 144.658,Z 473.768,A -85,B 0,C 180,E1 -33329.318,E2 -33329.318} C_VEL
LIN {X 0,Y 146.964,Z 467.205,A -85,B 0,C 180,E1 -33330.424,E2 -33330.424} C_VEL
LIN {X 0,Y 149.001,Z 460.385,A -85,B 0,C 180,E1 -33331.237,E2 -33331.237} C_VEL
LIN {X 0,Y 154.684,Z 452.696,A -85,B 0,C 180,E1 -33334.317,E2 -33334.317} C_VEL
LIN {X 0,Y 156.023,Z 450.771,A -85,B 0,C 180,E1 -33334.963,E2 -33334.963} C_VEL
LIN {X 0,Y 159.977,Z 448.169,A -85,B 0,C 180,E1 -33336.992,E2 -33336.992} C_VEL
LIN {X 0,Y 163.613,Z 444.922,A -85,B 0,C 180,E1 -33338.623,E2 -33338.623} C_VEL
LIN {X 0,Y 165.348,Z 444.74,A -85,B 0,C 180,E1 -33339.453,E2 -33339.453} C_VEL
LIN {X 0,Y 169.317,Z 453.334,A -85,B 0,C 180,E1 -33341.838,E2 -33341.838} C_VEL
LIN {X 0,Y 166.229,Z 498.485,A -85,B 0,C 180,E1 -33343.654,E2 -33343.654} C_VEL
LIN {X 0,Y 164.334,Z 513.044,A -85,B 0,C 180,E1 -33344.662,E2 -33344.662} C_VEL
LIN {X 0,Y 161.42,Z 527.224,A -85,B 0,C 180,E1 -33346.03,E2 -33346.03} C_VEL
LIN {X 0,Y 157.687,Z 540.705,A -85,B 0,C 180,E1 -33347.79,E2 -33347.79} C_VEL
LIN {X 0,Y 153.688,Z 552.791,A -85,B 0,C 180,E1 -33349.928,E2 -33349.928} C_VEL
LIN {X 0,Y 149.244,Z 563.896,A -85,B 0,C 180,E1 -33352.402,E2 -33352.402} C_VEL
LIN {X 0,Y 144.426,Z 574.147,A -85,B 0,C 180,E1 -33355.26,E2 -33355.26} C_VEL
LIN {X 0,Y 139.305,Z 583.843,A -85,B 0,C 180,E1 -33358.704,E2 -33358.704} C_VEL
LIN {X 0,Y 134.264,Z 592.778,A -85,B 0,C 180,E1 -33362.84,E2 -33362.84} C_VEL
LIN {X 0,Y 129.317,Z 600.858,A -85,B 0,C 180,E1 -33367.719,E2 -33367.719} C_VEL
LIN {X 0,Y 125.725,Z 606.524,A -85,B 0,C 180,E1 -33372.157,E2 -33372.157} C_VEL
LIN {X 0,Y 122.845,Z 611.172,A -85,B 0,C 180,E1 -33376.817,E2 -33376.817} C_VEL
LIN {X 0,Y 120.098,Z 616.003,A -85,B 0,C 180,E1 -33383.302,E2 -33383.302} C_VEL
LIN {X 0,Y 118.798,Z 619.372,A -85,B 0,C 180,E1 -33390.001,E2 -33390.001} C_VEL
LIN {X 0,Y 118.732,Z 621.41,A -85,B 0,C 180,E1 -33396.777,E2 -33396.777} C_VEL
LIN {X 0,Y 119.912,Z 622.156,A -85,B 0,C 180,E1 -33403.513,E2 -33403.513} C_VEL
LIN {X 0,Y 122.339,Z 621.612,A -85,B 0,C 180,E1 -33410.093,E2 -33410.093} C_VEL
LIN {X 0,Y 126.352,Z 619.716,A -85,B 0,C 180,E1 -33416.327,E2 -33416.327} C_VEL
LIN {X 0,Y 131.484,Z 616.458,A -85,B 0,C 180,E1 -33422.19,E2 -33422.19} C_VEL
LIN {X 0,Y 137.707,Z 611.72,A -85,B 0,C 180,E1 -33427.618,E2 -33427.618} C_VEL
LIN {X 0,Y 144.918,Z 605.352,A -85,B 0,C 180,E1 -33432.585,E2 -33432.585} C_VEL
LIN {X 0,Y 151.919,Z 598.221,A -85,B 0,C 180,E1 -33436.575,E2 -33436.575} C_VEL
LIN {X 0,Y 159.573,Z 589.339,A -85,B 0,C 180,E1 -33440.19,E2 -33440.19} C_VEL
LIN {X 0,Y 166.56,Z 579.977,A -85,B 0,C 180,E1 -33443.037,E2 -33443.037} C_VEL
LIN {X 0,Y 172.532,Z 570.511,A -85,B 0,C 180,E1 -33445.362,E2 -33445.362} C_VEL
LIN {X 0,Y 178.693,Z 559.334,A -85,B 0,C 180,E1 -33447.434,E2 -33447.434} C_VEL
LIN {X 0,Y 184.476,Z 546.761,A -85,B 0,C 180,E1 -33449.212,E2 -33449.212} C_VEL
LIN {X 0,Y 186.754,Z 540.838,A -85,B 0,C 180,E1 -33449.929,E2 -33449.929} C_VEL
LIN {X 0,Y 186.902,Z 539.813,A -85,B 0,C 180,E1 -33450.165,E2 -33450.165} C_VEL
LIN {X 0,Y 180.416,Z 546.575,A -85,B 0,C 180,E1 -33451.601,E2 -33451.601} C_VEL
LIN {X 0,Y 174.887,Z 551.503,A -85,B 0,C 180,E1 -33453.16,E2 -33453.16} C_VEL
LIN {X 0,Y 168.311,Z 557.938,A -85,B 0,C 180,E1 -33454.749,E2 -33454.749} C_VEL
LIN {X 0,Y 161.432,Z 563.639,A -85,B 0,C 180,E1 -33457.013,E2 -33457.013} C_VEL
LIN {X 0,Y 158.249,Z 565.963,A -85,B 0,C 180,E1 -33458.359,E2 -33458.359} C_VEL
LIN {X 0,Y 155.564,Z 567.916,A -85,B 0,C 180,E1 -33459.576,E2 -33459.576} C_VEL
LIN {X 0,Y 150.347,Z 572.189,A -85,B 0,C 180,E1 -33461.788,E2 -33461.788} C_VEL
LIN {X 0,Y 147.448,Z 574.268,A -85,B 0,C 180,E1 -33463.439,E2 -33463.439} C_VEL
LIN {X 0,Y 143.94,Z 576.743,A -85,B 0,C 180,E1 -33465.917,E2 -33465.917} C_VEL
LIN {X 0,Y 141.838,Z 578.537,A -85,B 0,C 180,E1 -33467.159,E2 -33467.159} C_VEL
LIN {X 0,Y 140.184,Z 579.795,A -85,B 0,C 180,E1 -33468.47,E2 -33468.47} C_VEL
LIN {X 0,Y 137.571,Z 581.765,A -85,B 0,C 180,E1 -33471.213,E2 -33471.213} C_VEL
LIN {X 0,Y 134.558,Z 584.552,A -85,B 0,C 180,E1 -33474.023,E2 -33474.023} C_VEL
LIN {X 0,Y 131.075,Z 588.332,A -85,B 0,C 180,E1 -33479.999,E2 -33479.999} C_VEL
LIN {X 0,Y 129.963,Z 589.736,A -85,B 0,C 180,E1 -33481.543,E2 -33481.543} C_VEL
LIN {X 0,Y 128.251,Z 594.307,A -85,B 0,C 180,E1 -33489.429,E2 -33489.429} C_VEL
LIN {X 0,Y 128.371,Z 595.946,A -85,B 0,C 180,E1 -33492.606,E2 -33492.606} C_VEL
LIN {X 0,Y 129.2,Z 597.272,A -85,B 0,C 180,E1 -33495.727,E2 -33495.727} C_VEL
LIN {X 0,Y 129.993,Z 599.005,A -85,B 0,C 180,E1 -33498.862,E2 -33498.862} C_VEL
LIN {X 0,Y 133.543,Z 601.627,A -85,B 0,C 180,E1 -33504.809,E2 -33504.809} C_VEL
LIN {X 0,Y 135.751,Z 603.028,A -85,B 0,C 180,E1 -33507.669,E2 -33507.669} C_VEL
LIN {X 0,Y 138.4,Z 603.25,A -85,B 0,C 180,E1 -33509.567,E2 -33509.567} C_VEL
LIN {X 0,Y 138.909,Z 603.448,A -85,B 0,C 180,E1 -33509.863,E2 -33509.863} C_VEL
LIN {X 0,Y 147.107,Z 612.293,A -85,B 0,C 180,E1 -33514.846,E2 -33514.846} C_VEL
LIN {X 0,Y 156.197,Z 619.327,A -85,B 0,C 180,E1 -33518.888,E2 -33518.888} C_VEL
LIN {X 0,Y 161.05,Z 622.405,A -85,B 0,C 180,E1 -33520.721,E2 -33520.721} C_VEL
LIN {X 0,Y 159.88,Z 622.467,A -85,B 0,C 180,E1 -33521.859,E2 -33521.859} C_VEL
LIN {X 0,Y 150.102,Z 619.63,A -85,B 0,C 180,E1 -33526.388,E2 -33526.388} C_VEL
LIN {X 0,Y 142.483,Z 626.383,A -85,B 0,C 180,E1 -33529.354,E2 -33529.354} C_VEL
LIN {X 0,Y 134.945,Z 632.742,A -85,B 0,C 180,E1 -33533.35,E2 -33533.35} C_VEL
LIN {X 0,Y 127.951,Z 638.478,A -85,B 0,C 180,E1 -33538.663,E2 -33538.663} C_VEL
LIN {X 0,Y 123.758,Z 641.781,A -85,B 0,C 180,E1 -33543.077,E2 -33543.077} C_VEL
LIN {X 0,Y 119.601,Z 645.016,A -85,B 0,C 180,E1 -33549.559,E2 -33549.559} C_VEL
LIN {X 0,Y 117.634,Z 646.873,A -85,B 0,C 180,E1 -33556.22,E2 -33556.22} C_VEL
LIN {X 0,Y 117.735,Z 647.526,A -85,B 0,C 180,E1 -33563.166,E2 -33563.166} C_VEL
LIN {X 0,Y 120.013,Z 646.939,A -85,B 0,C 180,E1 -33569.999,E2 -33569.999} C_VEL
LIN {X 0,Y 124.532,Z 645.119,A -85,B 0,C 180,E1 -33576.459,E2 -33576.459} C_VEL
LIN {X 0,Y 127.609,Z 643.702,A -85,B 0,C 180,E1 -33579.577,E2 -33579.577} C_VEL
LIN {X 0,Y 127.606,Z 651.085,A -85,B 0,C 180,E1 -33583.49,E2 -33583.49} C_VEL
LIN {X 0,Y 128.236,Z 660.017,A -85,B 0,C 180,E1 -33589.131,E2 -33589.131} C_VEL
LIN {X 0,Y 131.188,Z 669.8,A -85,B 0,C 180,E1 -33596.135,E2 -33596.135} C_VEL
LIN {X 0,Y 136.647,Z 678.155,A -85,B 0,C 180,E1 -33602.562,E2 -33602.562} C_VEL
LIN {X 0,Y 143.215,Z 684.468,A -85,B 0,C 180,E1 -33607.687,E2 -33607.687} C_VEL
LIN {X 0,Y 151.104,Z 689.835,A -85,B 0,C 180,E1 -33612.231,E2 -33612.231} C_VEL
LIN {X 0,Y 156.692,Z 692.756,A -85,B 0,C 180,E1 -33614.698,E2 -33614.698} C_VEL
LIN {X 0,Y 155.69,Z 692.249,A -85,B 0,C 180,E1 -33615.939,E2 -33615.939} C_VEL
LIN {X 0,Y 152.296,Z 690.436,A -85,B 0,C 180,E1 -33617.417,E2 -33617.417} C_VEL
LIN {X 0,Y 148.463,Z 688.217,A -85,B 0,C 180,E1 -33618.905,E2 -33618.905} C_VEL
LIN {X 0,Y 141.552,Z 683.656,A -85,B 0,C 180,E1 -33621.054,E2 -33621.054} C_VEL
LIN {X 0,Y 135.172,Z 678.655,A -85,B 0,C 180,E1 -33623.418,E2 -33623.418} C_VEL
LIN {X 0,Y 132.269,Z 675.779,A -85,B 0,C 180,E1 -33625.256,E2 -33625.256} C_VEL
LIN {X 0,Y 126.249,Z 667.081,A -85,B 0,C 180,E1 -33631.863,E2 -33631.863} C_VEL
LIN {X 0,Y 122.772,Z 657.274,A -85,B 0,C 180,E1 -33638.846,E2 -33638.846} C_VEL
LIN {X 0,Y 121.808,Z 649.156,A -85,B 0,C 180,E1 -33644.149,E2 -33644.149} C_VEL
LIN {X 0,Y 121.666,Z 641.153,A -85,B 0,C 180,E1 -33648.632,E2 -33648.632} C_VEL
LIN {X 0,Y 121.219,Z 634.142,A -85,B 0,C 180,E1 -33651.695,E2 -33651.695} C_VEL
LIN {X 0,Y 120.322,Z 622.446,A -85,B 0,C 180,E1 -33655.828,E2 -33655.828} C_VEL
LIN {X 0,Y 119.786,Z 610.94,A -85,B 0,C 180,E1 -33659.163,E2 -33659.163} C_VEL
LIN {X 0,Y 119.373,Z 595.648,A -85,B 0,C 180,E1 -33662.734,E2 -33662.734} C_VEL
LIN {X 0,Y 119.182,Z 581.536,A -85,B 0,C 180,E1 -33665.268,E2 -33665.268} C_VEL
LIN {X 0,Y 118.735,Z 554.272,A -85,B 0,C 180,E1 -33669.016,E2 -33669.016} C_VEL
LIN {X 0,Y 118.358,Z 537.903,A -85,B 0,C 180,E1 -33671.198,E2 -33671.198} C_VEL
LIN {X 0,Y 117.915,Z 539.526,A -85,B 0,C 180,E1 -33672.001,E2 -33672.001} C_VEL
LIN {X 0,Y 118.497,Z 539.252,A -85,B 0,C 180,E1 -33673.678,E2 -33673.678} C_VEL
LIN {X 0,Y 119.247,Z 538.002,A -85,B 0,C 180,E1 -33674.457,E2 -33674.457} C_VEL
LIN {X 0,Y 121.417,Z 533.886,A -85,B 0,C 180,E1 -33675.905,E2 -33675.905} C_VEL
LIN {X 0,Y 122.813,Z 530.844,A -85,B 0,C 180,E1 -33676.57,E2 -33676.57} C_VEL
LIN {X 0,Y 123.945,Z 529.721,A -85,B 0,C 180,E1 -33678.11,E2 -33678.11} C_VEL
LIN {X 0,Y 125.567,Z 527.337,A -85,B 0,C 180,E1 -33679.555,E2 -33679.555} C_VEL
LIN {X 0,Y 128.182,Z 522.261,A -85,B 0,C 180,E1 -33681.125,E2 -33681.125} C_VEL
LIN {X 0,Y 131.329,Z 514.471,A -85,B 0,C 180,E1 -33682.49,E2 -33682.49} C_VEL
LIN {X 0,Y 132.588,Z 511.145,A -85,B 0,C 180,E1 -33683.034,E2 -33683.034} C_VEL
LIN {X 0,Y 134.451,Z 508.272,A -85,B 0,C 180,E1 -33684.529,E2 -33684.529} C_VEL
LIN {X 0,Y 136.696,Z 503.649,A -85,B 0,C 180,E1 -33685.923,E2 -33685.923} C_VEL
LIN {X 0,Y 139.44,Z 495.77,A -85,B 0,C 180,E1 -33687.384,E2 -33687.384} C_VEL
LIN {X 0,Y 142.19,Z 486.468,A -85,B 0,C 180,E1 -33688.706,E2 -33688.706} C_VEL
LIN {X 0,Y 144.612,Z 482.554,A -85,B 0,C 180,E1 -33690.243,E2 -33690.243} C_VEL
LIN {X 0,Y 147.221,Z 476.928,A -85,B 0,C 180,E1 -33691.619,E2 -33691.619} C_VEL
LIN {X 0,Y 149.999,Z 469.195,A -85,B 0,C 180,E1 -33692.804,E2 -33692.804} C_VEL
LIN {X 0,Y 151.504,Z 464.567,A -85,B 0,C 180,E1 -33693.37,E2 -33693.37} C_VEL
LIN {X 0,Y 156.377,Z 458.297,A -85,B 0,C 180,E1 -33695.811,E2 -33695.811} C_VEL
LIN {X 0,Y 157.459,Z 456.937,A -85,B 0,C 180,E1 -33696.314,E2 -33696.314} C_VEL
LIN {X 0,Y 161.725,Z 453.968,A -85,B 0,C 180,E1 -33698.357,E2 -33698.357} C_VEL
LIN {X 0,Y 163.217,Z 452.616,A -85,B 0,C 180,E1 -33698.999,E2 -33698.999} C_VEL
LIN {X 0,Y 164.792,Z 456.043,A -85,B 0,C 180,E1 -33700.004,E2 -33700.004} C_VEL
LIN {X 0,Y 161.717,Z 499.06,A -85,B 0,C 180,E1 -33701.759,E2 -33701.759} C_VEL
LIN {X 0,Y 159.761,Z 513.43,A -85,B 0,C 180,E1 -33702.746,E2 -33702.746} C_VEL
LIN {X 0,Y 156.726,Z 527.706,A -85,B 0,C 180,E1 -33704.121,E2 -33704.121} C_VEL
LIN {X 0,Y 153.126,Z 540.376,A -85,B 0,C 180,E1 -33705.767,E2 -33705.767} C_VEL
LIN {X 0,Y 148.902,Z 552.679,A -85,B 0,C 180,E1 -33707.908,E2 -33707.908} C_VEL
LIN {X 0,Y 144.27,Z 563.932,A -85,B 0,C 180,E1 -33710.415,E2 -33710.415} C_VEL
LIN {X 0,Y 138.72,Z 575.266,A -85,B 0,C 180,E1 -33713.609,E2 -33713.609} C_VEL
LIN {X 0,Y 132.966,Z 585.569,A -85,B 0,C 180,E1 -33717.41,E2 -33717.41} C_VEL
LIN {X 0,Y 127.981,Z 593.876,A -85,B 0,C 180,E1 -33721.45,E2 -33721.45} C_VEL
LIN {X 0,Y 122.822,Z 601.809,A -85,B 0,C 180,E1 -33726.472,E2 -33726.472} C_VEL
LIN {X 0,Y 119.033,Z 607.456,A -85,B 0,C 180,E1 -33731.117,E2 -33731.117} C_VEL
LIN {X 0,Y 115.993,Z 612.068,A -85,B 0,C 180,E1 -33736.023,E2 -33736.023} C_VEL
LIN {X 0,Y 113.101,Z 616.866,A -85,B 0,C 180,E1 -33742.886,E2 -33742.886} C_VEL
LIN {X 0,Y 111.726,Z 620.208,A -85,B 0,C 180,E1 -33750.001,E2 -33750.001} C_VEL
LIN {X 0,Y 111.708,Z 622.214,A -85,B 0,C 180,E1 -33757.205,E2 -33757.205} C_VEL
LIN {X 0,Y 113.022,Z 622.927,A -85,B 0,C 180,E1 -33764.354,E2 -33764.354} C_VEL
LIN {X 0,Y 115.697,Z 622.347,A -85,B 0,C 180,E1 -33771.3,E2 -33771.3} C_VEL
LIN {X 0,Y 120.041,Z 620.419,A -85,B 0,C 180,E1 -33777.828,E2 -33777.828} C_VEL
LIN {X 0,Y 125.524,Z 617.132,A -85,B 0,C 180,E1 -33783.919,E2 -33783.919} C_VEL
LIN {X 0,Y 132.159,Z 612.36,A -85,B 0,C 180,E1 -33789.495,E2 -33789.495} C_VEL
LIN {X 0,Y 139.774,Z 605.957,A -85,B 0,C 180,E1 -33794.554,E2 -33794.554} C_VEL
LIN {X 0,Y 147.001,Z 598.906,A -85,B 0,C 180,E1 -33798.529,E2 -33798.529} C_VEL
LIN {X 0,Y 155.124,Z 589.836,A -85,B 0,C 180,E1 -33802.204,E2 -33802.204} C_VEL
LIN {X 0,Y 162.379,Z 580.42,A -85,B 0,C 180,E1 -33805.045,E2 -33805.045} C_VEL
LIN {X 0,Y 168.912,Z 570.374,A -85,B 0,C 180,E1 -33807.448,E2 -33807.448} C_VEL
LIN {X 0,Y 175.632,Z 558.344,A -85,B 0,C 180,E1 -33809.592,E2 -33809.592} C_VEL
LIN {X 0,Y 177.613,Z 554.352,A -85,B 0,C 180,E1 -33810.182,E2 -33810.182} C_VEL
LIN {X 0,Y 176.449,Z 554.432,A -85,B 0,C 180,E1 -33810.849,E2 -33810.849} C_VEL
LIN {X 0,Y 173.176,Z 557.297,A -85,B 0,C 180,E1 -33811.623,E2 -33811.623} C_VEL
LIN {X 0,Y 166.806,Z 562.954,A -85,B 0,C 180,E1 -33813.065,E2 -33813.065} C_VEL
LIN {X 0,Y 159.422,Z 568.549,A -85,B 0,C 180,E1 -33815.329,E2 -33815.329} C_VEL
LIN {X 0,Y 153.642,Z 572.416,A -85,B 0,C 180,E1 -33817.676,E2 -33817.676} C_VEL
LIN {X 0,Y 149.15,Z 575.828,A -85,B 0,C 180,E1 -33819.375,E2 -33819.375} C_VEL
LIN {X 0,Y 144.58,Z 578.914,A -85,B 0,C 180,E1 -33821.644,E2 -33821.644} C_VEL
LIN {X 0,Y 141.066,Z 581.144,A -85,B 0,C 180,E1 -33823.948,E2 -33823.948} C_VEL
LIN {X 0,Y 138.588,Z 583.022,A -85,B 0,C 180,E1 -33825.361,E2 -33825.361} C_VEL
LIN {X 0,Y 135.221,Z 585.322,A -85,B 0,C 180,E1 -33828.041,E2 -33828.041} C_VEL
LIN {X 0,Y 132.286,Z 587.474,A -85,B 0,C 180,E1 -33830.859,E2 -33830.859} C_VEL
LIN {X 0,Y 129.309,Z 590.012,A -85,B 0,C 180,E1 -33833.78,E2 -33833.78} C_VEL
LIN {X 0,Y 126.098,Z 593.152,A -85,B 0,C 180,E1 -33839.081,E2 -33839.081} C_VEL
LIN {X 0,Y 125.401,Z 593.923,A -85,B 0,C 180,E1 -33839.999,E2 -33839.999} C_VEL
LIN {X 0,Y 122.761,Z 599.443,A -85,B 0,C 180,E1 -33849.855,E2 -33849.855} C_VEL
LIN {X 0,Y 123.912,Z 602.221,A -85,B 0,C 180,E1 -33856.417,E2 -33856.417} C_VEL
LIN {X 0,Y 124.88,Z 603.796,A -85,B 0,C 180,E1 -33859.665,E2 -33859.665} C_VEL
LIN {X 0,Y 131.009,Z 607.639,A -85,B 0,C 180,E1 -33868.762,E2 -33868.762} C_VEL
LIN {X 0,Y 134.2,Z 608.464,A -85,B 0,C 180,E1 -33871.462,E2 -33871.462} C_VEL
LIN {X 0,Y 137.213,Z 609.737,A -85,B 0,C 180,E1 -33874.161,E2 -33874.161} C_VEL
LIN {X 0,Y 141.235,Z 609.993,A -85,B 0,C 180,E1 -33876.3,E2 -33876.3} C_VEL
LIN {X 0,Y 152.312,Z 618.596,A -85,B 0,C 180,E1 -33881.12,E2 -33881.12} C_VEL
LIN {X 0,Y 150.915,Z 618.343,A -85,B 0,C 180,E1 -33882.045,E2 -33882.045} C_VEL
LIN {X 0,Y 147.318,Z 617.09,A -85,B 0,C 180,E1 -33883.77,E2 -33883.77} C_VEL
LIN {X 0,Y 139.623,Z 623.754,A -85,B 0,C 180,E1 -33886.385,E2 -33886.385} C_VEL
LIN {X 0,Y 131.417,Z 630.469,A -85,B 0,C 180,E1 -33890.238,E2 -33890.238} C_VEL
LIN {X 0,Y 125.445,Z 635.156,A -85,B 0,C 180,E1 -33894.105,E2 -33894.105} C_VEL
LIN {X 0,Y 118.848,Z 640.098,A -85,B 0,C 180,E1 -33899.936,E2 -33899.936} C_VEL
LIN {X 0,Y 115.014,Z 642.832,A -85,B 0,C 180,E1 -33904.766,E2 -33904.766} C_VEL
LIN {X 0,Y 111.565,Z 645.336,A -85,B 0,C 180,E1 -33911.704,E2 -33911.704} C_VEL
LIN {X 0,Y 110.347,Z 646.58,A -85,B 0,C 180,E1 -33919.021,E2 -33919.021} C_VEL
LIN {X 0,Y 111.418,Z 646.584,A -85,B 0,C 180,E1 -33926.395,E2 -33926.395} C_VEL
LIN {X 0,Y 114.778,Z 645.35,A -85,B 0,C 180,E1 -33933.498,E2 -33933.498} C_VEL
LIN {X 0,Y 120.328,Z 642.853,A -85,B 0,C 180,E1 -33940.057,E2 -33940.057} C_VEL
LIN {X 0,Y 121.97,Z 642.156,A -85,B 0,C 180,E1 -33941.7,E2 -33941.7} C_VEL
LIN {X 0,Y 122.151,Z 650.792,A -85,B 0,C 180,E1 -33946.661,E2 -33946.661} C_VEL
LIN {X 0,Y 123.717,Z 660.663,A -85,B 0,C 180,E1 -33953.348,E2 -33953.348} C_VEL
LIN {X 0,Y 127.296,Z 669.155,A -85,B 0,C 180,E1 -33959.684,E2 -33959.684} C_VEL
LIN {X 0,Y 132.896,Z 676.628,A -85,B 0,C 180,E1 -33965.434,E2 -33965.434} C_VEL
LIN {X 0,Y 140.058,Z 683.062,A -85,B 0,C 180,E1 -33970.552,E2 -33970.552} C_VEL
LIN {X 0,Y 148.542,Z 688.524,A -85,B 0,C 180,E1 -33975.017,E2 -33975.017} C_VEL
LIN {X 0,Y 144.313,Z 685.961,A -85,B 0,C 180,E1 -33977.195,E2 -33977.195} C_VEL
LIN {X 0,Y 136.446,Z 679.989,A -85,B 0,C 180,E1 -33981.975,E2 -33981.975} C_VEL
LIN {X 0,Y 132.269,Z 675.779,A -85,B 0,C 180,E1 -33985.256,E2 -33985.256} C_VEL
LIN {X 0,Y 129.619,Z 672.839,A -85,B 0,C 180,E1 -33987.154,E2 -33987.154} C_VEL
LIN {X 0,Y 124.562,Z 666.97,A -85,B 0,C 180,E1 -33989.922,E2 -33989.922} C_VEL
LIN {X 0,Y 120.068,Z 660.616,A -85,B 0,C 180,E1 -33992.852,E2 -33992.852} C_VEL
LIN {X 0,Y 118.413,Z 657.051,A -85,B 0,C 180,E1 -33994.997,E2 -33994.997} C_VEL
LIN {X 0,Y 116.443,Z 645.987,A -85,B 0,C 180,E1 -34002.497,E2 -34002.497} C_VEL
LIN {X 0,Y 116.132,Z 637.117,A -85,B 0,C 180,E1 -34007.557,E2 -34007.557} C_VEL
LIN {X 0,Y 115.367,Z 628.856,A -85,B 0,C 180,E1 -34011.05,E2 -34011.05} C_VEL
LIN {X 0,Y 114.387,Z 616.854,A -85,B 0,C 180,E1 -34015.171,E2 -34015.171} C_VEL
LIN {X 0,Y 113.741,Z 606.026,A -85,B 0,C 180,E1 -34018.236,E2 -34018.236} C_VEL
LIN {X 0,Y 113.261,Z 590.612,A -85,B 0,C 180,E1 -34021.773,E2 -34021.773} C_VEL
LIN {X 0,Y 112.989,Z 575.823,A -85,B 0,C 180,E1 -34024.335,E2 -34024.335} C_VEL
LIN {X 0,Y 112.244,Z 550.487,A -85,B 0,C 180,E1 -34027.96,E2 -34027.96} C_VEL
LIN {X 0,Y 111.61,Z 551.97,A -85,B 0,C 180,E1 -34029.028,E2 -34029.028} C_VEL
LIN {X 0,Y 112.104,Z 551.494,A -85,B 0,C 180,E1 -34030.805,E2 -34030.805} C_VEL
LIN {X 0,Y 112.938,Z 550.174,A -85,B 0,C 180,E1 -34031.72,E2 -34031.72} C_VEL
LIN {X 0,Y 115.111,Z 546.529,A -85,B 0,C 180,E1 -34033.199,E2 -34033.199} C_VEL
LIN {X 0,Y 115.719,Z 545.748,A -85,B 0,C 180,E1 -34034.013,E2 -34034.013} C_VEL
LIN {X 0,Y 116.723,Z 544.767,A -85,B 0,C 180,E1 -34035.668,E2 -34035.668} C_VEL
LIN {X 0,Y 118.491,Z 542.202,A -85,B 0,C 180,E1 -34037.193,E2 -34037.193} C_VEL
LIN {X 0,Y 122.113,Z 536.13,A -85,B 0,C 180,E1 -34039.259,E2 -34039.259} C_VEL
LIN {X 0,Y 124.127,Z 533.81,A -85,B 0,C 180,E1 -34041.113,E2 -34041.113} C_VEL
LIN {X 0,Y 126.765,Z 529.851,A -85,B 0,C 180,E1 -34042.756,E2 -34042.756} C_VEL
LIN {X 0,Y 130.24,Z 523.358,A -85,B 0,C 180,E1 -34044.323,E2 -34044.323} C_VEL
LIN {X 0,Y 133.439,Z 515.909,A -85,B 0,C 180,E1 -34045.454,E2 -34045.454} C_VEL
LIN {X 0,Y 136.422,Z 511.34,A -85,B 0,C 180,E1 -34047.316,E2 -34047.316} C_VEL
LIN {X 0,Y 139.45,Z 505.015,A -85,B 0,C 180,E1 -34048.81,E2 -34048.81} C_VEL
LIN {X 0,Y 142.869,Z 495.451,A -85,B 0,C 180,E1 -34050.27,E2 -34050.27} C_VEL
LIN {X 0,Y 144.359,Z 490.852,A -85,B 0,C 180,E1 -34050.933,E2 -34050.933} C_VEL
LIN {X 0,Y 147.456,Z 485.624,A -85,B 0,C 180,E1 -34052.649,E2 -34052.649} C_VEL
LIN {X 0,Y 150.81,Z 478.14,A -85,B 0,C 180,E1 -34054.171,E2 -34054.171} C_VEL
LIN {X 0,Y 153.934,Z 469.196,A -85,B 0,C 180,E1 -34055.305,E2 -34055.305} C_VEL
LIN {X 0,Y 158.845,Z 463.162,A -85,B 0,C 180,E1 -34057.574,E2 -34057.574} C_VEL
LIN {X 0,Y 160.118,Z 462.365,A -85,B 0,C 180,E1 -34058.178,E2 -34058.178} C_VEL
LIN {X 0,Y 157.359,Z 499.783,A -85,B 0,C 180,E1 -34059.759,E2 -34059.759} C_VEL
LIN {X 0,Y 155.378,Z 513.815,A -85,B 0,C 180,E1 -34060.72,E2 -34060.72} C_VEL
LIN {X 0,Y 152.548,Z 527.063,A -85,B 0,C 180,E1 -34061.99,E2 -34061.99} C_VEL
LIN {X 0,Y 148.756,Z 540.05,A -85,B 0,C 180,E1 -34063.618,E2 -34063.618} C_VEL
LIN {X 0,Y 144.325,Z 552.563,A -85,B 0,C 180,E1 -34065.761,E2 -34065.761} C_VEL
LIN {X 0,Y 139.456,Z 563.974,A -85,B 0,C 180,E1 -34068.279,E2 -34068.279} C_VEL
LIN {X 0,Y 134.156,Z 574.466,A -85,B 0,C 180,E1 -34071.206,E2 -34071.206} C_VEL
LIN {X 0,Y 128.143,Z 584.885,A -85,B 0,C 180,E1 -34074.975,E2 -34074.975} C_VEL
LIN {X 0,Y 122.732,Z 593.476,A -85,B 0,C 180,E1 -34079.094,E2 -34079.094} C_VEL
LIN {X 0,Y 117.906,Z 600.626,A -85,B 0,C 180,E1 -34083.542,E2 -34083.542} C_VEL
LIN {X 0,Y 113.618,Z 606.607,A -85,B 0,C 180,E1 -34088.291,E2 -34088.291} C_VEL
LIN {X 0,Y 109.167,Z 612.964,A -85,B 0,C 180,E1 -34095.129,E2 -34095.129} C_VEL
LIN {X 0,Y 106.126,Z 617.728,A -85,B 0,C 180,E1 -34102.415,E2 -34102.415} C_VEL
LIN {X 0,Y 104.682,Z 621.04,A -85,B 0,C 180,E1 -34110.001,E2 -34110.001} C_VEL
LIN {X 0,Y 104.704,Z 623.012,A -85,B 0,C 180,E1 -34117.69,E2 -34117.69} C_VEL
LIN {X 0,Y 106.17,Z 623.692,A -85,B 0,C 180,E1 -34125.302,E2 -34125.302} C_VEL
LIN {X 0,Y 109.116,Z 623.081,A -85,B 0,C 180,E1 -34132.654,E2 -34132.654} C_VEL
LIN {X 0,Y 113.807,Z 621.124,A -85,B 0,C 180,E1 -34139.498,E2 -34139.498} C_VEL
LIN {X 0,Y 119.695,Z 617.805,A -85,B 0,C 180,E1 -34145.817,E2 -34145.817} C_VEL
LIN {X 0,Y 126.755,Z 613.001,A -85,B 0,C 180,E1 -34151.539,E2 -34151.539} C_VEL
LIN {X 0,Y 132.697,Z 608.331,A -85,B 0,C 180,E1 -34155.448,E2 -34155.448} C_VEL
LIN {X 0,Y 139.498,Z 602.267,A -85,B 0,C 180,E1 -34159.249,E2 -34159.249} C_VEL
LIN {X 0,Y 147.232,Z 594.429,A -85,B 0,C 180,E1 -34162.833,E2 -34162.833} C_VEL
LIN {X 0,Y 154.651,Z 585.823,A -85,B 0,C 180,E1 -34165.75,E2 -34165.75} C_VEL
LIN {X 0,Y 162.122,Z 575.491,A -85,B 0,C 180,E1 -34168.504,E2 -34168.504} C_VEL
LIN {X 0,Y 167.314,Z 567.346,A -85,B 0,C 180,E1 -34170.186,E2 -34170.186} C_VEL
LIN {X 0,Y 167.801,Z 565.803,A -85,B 0,C 180,E1 -34170.719,E2 -34170.719} C_VEL
LIN {X 0,Y 160.846,Z 570.922,A -85,B 0,C 180,E1 -34172.48,E2 -34172.48} C_VEL
LIN {X 0,Y 154.663,Z 575.014,A -85,B 0,C 180,E1 -34174.515,E2 -34174.515} C_VEL
LIN {X 0,Y 152.16,Z 576.478,A -85,B 0,C 180,E1 -34175.524,E2 -34175.524} C_VEL
LIN {X 0,Y 143.958,Z 581.994,A -85,B 0,C 180,E1 -34178.604,E2 -34178.604} C_VEL
LIN {X 0,Y 137.605,Z 585.717,A -85,B 0,C 180,E1 -34182.216,E2 -34182.216} C_VEL
LIN {X 0,Y 135.278,Z 587.317,A -85,B 0,C 180,E1 -34183.453,E2 -34183.453} C_VEL
LIN {X 0,Y 131.594,Z 589.609,A -85,B 0,C 180,E1 -34186.124,E2 -34186.124} C_VEL
LIN {X 0,Y 128.478,Z 591.625,A -85,B 0,C 180,E1 -34188.917,E2 -34188.917} C_VEL
LIN {X 0,Y 125.121,Z 594.146,A -85,B 0,C 180,E1 -34191.954,E2 -34191.954} C_VEL
LIN {X 0,Y 121.047,Z 597.612,A -85,B 0,C 180,E1 -34197.963,E2 -34197.963} C_VEL
LIN {X 0,Y 118.5,Z 600.697,A -85,B 0,C 180,E1 -34203.388,E2 -34203.388} C_VEL
LIN {X 0,Y 117.246,Z 604.125,A -85,B 0,C 180,E1 -34210.324,E2 -34210.324} C_VEL
LIN {X 0,Y 119.595,Z 608.318,A -85,B 0,C 180,E1 -34220.573,E2 -34220.573} C_VEL
LIN {X 0,Y 126.106,Z 612.02,A -85,B 0,C 180,E1 -34229.992,E2 -34229.992} C_VEL
LIN {X 0,Y 129.341,Z 612.919,A -85,B 0,C 180,E1 -34232.788,E2 -34232.788} C_VEL
LIN {X 0,Y 132.598,Z 614.052,A -85,B 0,C 180,E1 -34235.525,E2 -34235.525} C_VEL
LIN {X 0,Y 136.89,Z 614.506,A -85,B 0,C 180,E1 -34237.88,E2 -34237.88} C_VEL
LIN {X 0,Y 141.853,Z 615.755,A -85,B 0,C 180,E1 -34240.875,E2 -34240.875} C_VEL
LIN {X 0,Y 142.295,Z 616.678,A -85,B 0,C 180,E1 -34241.748,E2 -34241.748} C_VEL
LIN {X 0,Y 134.601,Z 623.168,A -85,B 0,C 180,E1 -34244.312,E2 -34244.312} C_VEL
LIN {X 0,Y 126.059,Z 629.841,A -85,B 0,C 180,E1 -34248.18,E2 -34248.18} C_VEL
LIN {X 0,Y 119.776,Z 634.507,A -85,B 0,C 180,E1 -34252.117,E2 -34252.117} C_VEL
LIN {X 0,Y 112.742,Z 639.415,A -85,B 0,C 180,E1 -34258.123,E2 -34258.123} C_VEL
LIN {X 0,Y 108.616,Z 642.12,A -85,B 0,C 180,E1 -34263.165,E2 -34263.165} C_VEL
LIN {X 0,Y 104.813,Z 644.594,A -85,B 0,C 180,E1 -34270.479,E2 -34270.479} C_VEL
LIN {X 0,Y 103.311,Z 645.807,A -85,B 0,C 180,E1 -34278.264,E2 -34278.264} C_VEL
LIN {X 0,Y 104.247,Z 645.782,A -85,B 0,C 180,E1 -34286.147,E2 -34286.147} C_VEL
LIN {X 0,Y 107.544,Z 644.512,A -85,B 0,C 180,E1 -34293.734,E2 -34293.734} C_VEL
LIN {X 0,Y 113.197,Z 641.987,A -85,B 0,C 180,E1 -34300.698,E2 -34300.698} C_VEL
LIN {X 0,Y 116.529,Z 640.266,A -85,B 0,C 180,E1 -34303.912,E2 -34303.912} C_VEL
LIN {X 0,Y 116.922,Z 649.021,A -85,B 0,C 180,E1 -34309.237,E2 -34309.237} C_VEL
LIN {X 0,Y 119.334,Z 659.537,A -85,B 0,C 180,E1 -34316.645,E2 -34316.645} C_VEL
LIN {X 0,Y 123.326,Z 667.456,A -85,B 0,C 180,E1 -34322.653,E2 -34322.653} C_VEL
LIN {X 0,Y 129.563,Z 674.975,A -85,B 0,C 180,E1 -34328.441,E2 -34328.441} C_VEL
LIN {X 0,Y 139.42,Z 682.975,A -85,B 0,C 180,E1 -34334.697,E2 -34334.697} C_VEL
LIN {X 0,Y 139.621,Z 683.11,A -85,B 0,C 180,E1 -34335.385,E2 -34335.385} C_VEL
LIN {X 0,Y 129.693,Z 675.018,A -85,B 0,C 180,E1 -34341.605,E2 -34341.605} C_VEL
LIN {X 0,Y 122.714,Z 666.367,A -85,B 0,C 180,E1 -34348.131,E2 -34348.131} C_VEL
LIN {X 0,Y 118.413,Z 657.051,A -85,B 0,C 180,E1 -34354.997,E2 -34354.997} C_VEL
LIN {X 0,Y 117.079,Z 653.494,A -85,B 0,C 180,E1 -34357.178,E2 -34357.178} C_VEL
LIN {X 0,Y 114.244,Z 646.533,A -85,B 0,C 180,E1 -34360.348,E2 -34360.348} C_VEL
LIN {X 0,Y 111.243,Z 637.513,A -85,B 0,C 180,E1 -34364.104,E2 -34364.104} C_VEL
LIN {X 0,Y 110.817,Z 634.578,A -85,B 0,C 180,E1 -34365.493,E2 -34365.493} C_VEL
LIN {X 0,Y 110.198,Z 628.539,A -85,B 0,C 180,E1 -34368.221,E2 -34368.221} C_VEL
LIN {X 0,Y 108.944,Z 616.604,A -85,B 0,C 180,E1 -34372.613,E2 -34372.613} C_VEL
LIN {X 0,Y 108.167,Z 605.944,A -85,B 0,C 180,E1 -34375.823,E2 -34375.823} C_VEL
LIN {X 0,Y 107.434,Z 590.78,A -85,B 0,C 180,E1 -34379.534,E2 -34379.534} C_VEL
LIN {X 0,Y 106.976,Z 576.241,A -85,B 0,C 180,E1 -34382.239,E2 -34382.239} C_VEL
LIN {X 0,Y 106.384,Z 561.159,A -85,B 0,C 180,E1 -34384.656,E2 -34384.656} C_VEL
LIN {X 0,Y 106.042,Z 561.69,A -85,B 0,C 180,E1 -34384.96,E2 -34384.96} C_VEL
LIN {X 0,Y 105.614,Z 562.343,A -85,B 0,C 180,E1 -34385.841,E2 -34385.841} C_VEL
LIN {X 0,Y 106.078,Z 561.647,A -85,B 0,C 180,E1 -34387.922,E2 -34387.922} C_VEL
LIN {X 0,Y 107.475,Z 559.555,A -85,B 0,C 180,E1 -34389.376,E2 -34389.376} C_VEL
LIN {X 0,Y 108.759,Z 557.738,A -85,B 0,C 180,E1 -34391.141,E2 -34391.141} C_VEL
LIN {X 0,Y 109.669,Z 556.744,A -85,B 0,C 180,E1 -34392.918,E2 -34392.918} C_VEL
LIN {X 0,Y 111.457,Z 554.312,A -85,B 0,C 180,E1 -34394.56,E2 -34394.56} C_VEL
LIN {X 0,Y 112.71,Z 552.531,A -85,B 0,C 180,E1 -34395.386,E2 -34395.386} C_VEL
LIN {X 0,Y 113.695,Z 551.259,A -85,B 0,C 180,E1 -34396.236,E2 -34396.236} C_VEL
LIN {X 0,Y 114.868,Z 550.139,A -85,B 0,C 180,E1 -34397.753,E2 -34397.753} C_VEL
LIN {X 0,Y 117.886,Z 546.3,A -85,B 0,C 180,E1 -34399.978,E2 -34399.978} C_VEL
LIN {X 0,Y 121.036,Z 541.599,A -85,B 0,C 180,E1 -34401.539,E2 -34401.539} C_VEL
LIN {X 0,Y 123.507,Z 538.887,A -85,B 0,C 180,E1 -34403.391,E2 -34403.391} C_VEL
LIN {X 0,Y 127.168,Z 533.91,A -85,B 0,C 180,E1 -34405.378,E2 -34405.378} C_VEL
LIN {X 0,Y 130.534,Z 528.367,A -85,B 0,C 180,E1 -34406.706,E2 -34406.706} C_VEL
LIN {X 0,Y 134.649,Z 520.131,A -85,B 0,C 180,E1 -34408.012,E2 -34408.012} C_VEL
LIN {X 0,Y 138.225,Z 514.853,A -85,B 0,C 180,E1 -34409.818,E2 -34409.818} C_VEL
LIN {X 0,Y 141.595,Z 508.407,A -85,B 0,C 180,E1 -34411.191,E2 -34411.191} C_VEL
LIN {X 0,Y 145.473,Z 498.504,A -85,B 0,C 180,E1 -34412.594,E2 -34412.594} C_VEL
LIN {X 0,Y 146.617,Z 495.305,A -85,B 0,C 180,E1 -34413.02,E2 -34413.02} C_VEL
LIN {X 0,Y 150.409,Z 488.84,A -85,B 0,C 180,E1 -34414.886,E2 -34414.886} C_VEL
LIN {X 0,Y 153.95,Z 480.983,A -85,B 0,C 180,E1 -34416.32,E2 -34416.32} C_VEL
LIN {X 0,Y 155.009,Z 478.284,A -85,B 0,C 180,E1 -34416.698,E2 -34416.698} C_VEL
LIN {X 0,Y 153.083,Z 501.586,A -85,B 0,C 180,E1 -34417.72,E2 -34417.72} C_VEL
LIN {X 0,Y 150.934,Z 515.682,A -85,B 0,C 180,E1 -34418.72,E2 -34418.72} C_VEL
LIN {X 0,Y 147.9,Z 528.672,A -85,B 0,C 180,E1 -34419.948,E2 -34419.948} C_VEL
LIN {X 0,Y 144.011,Z 541.459,A -85,B 0,C 180,E1 -34421.599,E2 -34421.599} C_VEL
LIN {X 0,Y 139.403,Z 553.844,A -85,B 0,C 180,E1 -34423.757,E2 -34423.757} C_VEL
LIN {X 0,Y 134.301,Z 565.166,A -85,B 0,C 180,E1 -34426.287,E2 -34426.287} C_VEL
LIN {X 0,Y 128.761,Z 575.586,A -85,B 0,C 180,E1 -34429.248,E2 -34429.248} C_VEL
LIN {X 0,Y 122.465,Z 585.945,A -85,B 0,C 180,E1 -34433.091,E2 -34433.091} C_VEL
LIN {X 0,Y 116.753,Z 594.488,A -85,B 0,C 180,E1 -34437.321,E2 -34437.321} C_VEL
LIN {X 0,Y 111.64,Z 601.597,A -85,B 0,C 180,E1 -34441.93,E2 -34441.93} C_VEL
LIN {X 0,Y 107.102,Z 607.538,A -85,B 0,C 180,E1 -34446.897,E2 -34446.897} C_VEL
LIN {X 0,Y 102.373,Z 613.861,A -85,B 0,C 180,E1 -34454.117,E2 -34454.117} C_VEL
LIN {X 0,Y 99.147,Z 618.591,A -85,B 0,C 180,E1 -34461.878,E2 -34461.878} C_VEL
LIN {X 0,Y 97.613,Z 621.872,A -85,B 0,C 180,E1 -34470.001,E2 -34470.001} C_VEL
LIN {X 0,Y 97.692,Z 623.808,A -85,B 0,C 180,E1 -34478.245,E2 -34478.245} C_VEL
LIN {X 0,Y 99.357,Z 624.454,A -85,B 0,C 180,E1 -34486.38,E2 -34486.38} C_VEL
LIN {X 0,Y 102.606,Z 623.815,A -85,B 0,C 180,E1 -34494.18,E2 -34494.18} C_VEL
LIN {X 0,Y 107.685,Z 621.829,A -85,B 0,C 180,E1 -34501.358,E2 -34501.358} C_VEL
LIN {X 0,Y 114.017,Z 618.478,A -85,B 0,C 180,E1 -34507.904,E2 -34507.904} C_VEL
LIN {X 0,Y 121.53,Z 613.641,A -85,B 0,C 180,E1 -34513.76,E2 -34513.76} C_VEL
LIN {X 0,Y 127.821,Z 608.935,A -85,B 0,C 180,E1 -34517.714,E2 -34517.714} C_VEL
LIN {X 0,Y 135.739,Z 602.118,A -85,B 0,C 180,E1 -34521.901,E2 -34521.901} C_VEL
LIN {X 0,Y 144.311,Z 593.616,A -85,B 0,C 180,E1 -34525.603,E2 -34525.603} C_VEL
LIN {X 0,Y 152.062,Z 584.688,A -85,B 0,C 180,E1 -34528.449,E2 -34528.449} C_VEL
LIN {X 0,Y 157.604,Z 577.24,A -85,B 0,C 180,E1 -34530.39,E2 -34530.39} C_VEL
LIN {X 0,Y 158.226,Z 575.978,A -85,B 0,C 180,E1 -34530.858,E2 -34530.858} C_VEL
LIN {X 0,Y 147.787,Z 582.221,A -85,B 0,C 180,E1 -34534.227,E2 -34534.227} C_VEL
LIN {X 0,Y 141.196,Z 586.25,A -85,B 0,C 180,E1 -34536.617,E2 -34536.617} C_VEL
LIN {X 0,Y 133.721,Z 590.294,A -85,B 0,C 180,E1 -34540.539,E2 -34540.539} C_VEL
LIN {X 0,Y 129.812,Z 592.644,A -85,B 0,C 180,E1 -34542.735,E2 -34542.735} C_VEL
LIN {X 0,Y 124.46,Z 595.681,A -85,B 0,C 180,E1 -34546.989,E2 -34546.989} C_VEL
LIN {X 0,Y 120.895,Z 598.055,A -85,B 0,C 180,E1 -34549.989,E2 -34549.989} C_VEL
LIN {X 0,Y 112.692,Z 605.303,A -85,B 0,C 180,E1 -34563.563,E2 -34563.563} C_VEL
LIN {X 0,Y 111.539,Z 608.525,A -85,B 0,C 180,E1 -34570.858,E2 -34570.858} C_VEL
LIN {X 0,Y 116.163,Z 613.904,A -85,B 0,C 180,E1 -34585.246,E2 -34585.246} C_VEL
LIN {X 0,Y 121.085,Z 616.134,A -85,B 0,C 180,E1 -34591.373,E2 -34591.373} C_VEL
LIN {X 0,Y 127.908,Z 618.099,A -85,B 0,C 180,E1 -34597.039,E2 -34597.039} C_VEL
LIN {X 0,Y 132.279,Z 618.641,A -85,B 0,C 180,E1 -34599.451,E2 -34599.451} C_VEL
LIN {X 0,Y 133.201,Z 619.833,A -85,B 0,C 180,E1 -34600.9,E2 -34600.9} C_VEL
LIN {X 0,Y 125.806,Z 625.596,A -85,B 0,C 180,E1 -34603.63,E2 -34603.63} C_VEL
LIN {X 0,Y 118.602,Z 630.849,A -85,B 0,C 180,E1 -34607.22,E2 -34607.22} C_VEL
LIN {X 0,Y 110.31,Z 636.482,A -85,B 0,C 180,E1 -34612.898,E2 -34612.898} C_VEL
LIN {X 0,Y 105.17,Z 639.69,A -85,B 0,C 180,E1 -34617.804,E2 -34617.804} C_VEL
LIN {X 0,Y 99.938,Z 642.792,A -85,B 0,C 180,E1 -34625.131,E2 -34625.131} C_VEL
LIN {X 0,Y 96.92,Z 644.601,A -85,B 0,C 180,E1 -34633.196,E2 -34633.196} C_VEL
LIN {X 0,Y 96.372,Z 645.162,A -85,B 0,C 180,E1 -34641.641,E2 -34641.641} C_VEL
LIN {X 0,Y 98.365,Z 644.481,A -85,B 0,C 180,E1 -34649.999,E2 -34649.999} C_VEL
LIN {X 0,Y 102.924,Z 642.561,A -85,B 0,C 180,E1 -34657.822,E2 -34657.822} C_VEL
LIN {X 0,Y 109.5,Z 639.313,A -85,B 0,C 180,E1 -34664.825,E2 -34664.825} C_VEL
LIN {X 0,Y 111.279,Z 638.428,A -85,B 0,C 180,E1 -34666.425,E2 -34666.425} C_VEL
LIN {X 0,Y 112.25,Z 648.429,A -85,B 0,C 180,E1 -34672.954,E2 -34672.954} C_VEL
LIN {X 0,Y 115.458,Z 658.458,A -85,B 0,C 180,E1 -34680.329,E2 -34680.329} C_VEL
LIN {X 0,Y 121.365,Z 667.655,A -85,B 0,C 180,E1 -34687.3,E2 -34687.3} C_VEL
LIN {X 0,Y 130.666,Z 676.664,A -85,B 0,C 180,E1 -34694.176,E2 -34694.176} C_VEL
LIN {X 0,Y 131.722,Z 677.479,A -85,B 0,C 180,E1 -34694.807,E2 -34694.807} C_VEL
LIN {X 0,Y 130.803,Z 676.761,A -85,B 0,C 180,E1 -34695.883,E2 -34695.883} C_VEL
LIN {X 0,Y 123.132,Z 669.596,A -85,B 0,C 180,E1 -34701.264,E2 -34701.264} C_VEL
LIN {X 0,Y 117.052,Z 661.369,A -85,B 0,C 180,E1 -34707.415,E2 -34707.415} C_VEL
LIN {X 0,Y 112.639,Z 650.729,A -85,B 0,C 180,E1 -34715.182,E2 -34715.182} C_VEL
LIN {X 0,Y 111.144,Z 641.163,A -85,B 0,C 180,E1 -34721.634,E2 -34721.634} C_VEL
LIN {X 0,Y 110.817,Z 634.578,A -85,B 0,C 180,E1 -34725.493,E2 -34725.493} C_VEL
LIN {X 0,Y 110.317,Z 631.597,A -85,B 0,C 180,E1 -34726.769,E2 -34726.769} C_VEL
LIN {X 0,Y 109.425,Z 628.369,A -85,B 0,C 180,E1 -34727.825,E2 -34727.825} C_VEL
LIN {X 0,Y 106.988,Z 621.528,A -85,B 0,C 180,E1 -34729.483,E2 -34729.483} C_VEL
LIN {X 0,Y 104.438,Z 614.259,A -85,B 0,C 180,E1 -34730.957,E2 -34730.957} C_VEL
LIN {X 0,Y 103.111,Z 608.795,A -85,B 0,C 180,E1 -34732.244,E2 -34732.244} C_VEL
LIN {X 0,Y 102.908,Z 606.992,A -85,B 0,C 180,E1 -34732.755,E2 -34732.755} C_VEL
LIN {X 0,Y 101.835,Z 591.785,A -85,B 0,C 180,E1 -34736.797,E2 -34736.797} C_VEL
LIN {X 0,Y 101.273,Z 577.902,A -85,B 0,C 180,E1 -34739.63,E2 -34739.63} C_VEL
LIN {X 0,Y 100.904,Z 570.384,A -85,B 0,C 180,E1 -34740.871,E2 -34740.871} C_VEL
LIN {X 0,Y 99.917,Z 571.552,A -85,B 0,C 180,E1 -34742.01,E2 -34742.01} C_VEL
LIN {X 0,Y 99.884,Z 571.26,A -85,B 0,C 180,E1 -34744.022,E2 -34744.022} C_VEL
LIN {X 0,Y 100.356,Z 570.476,A -85,B 0,C 180,E1 -34744.919,E2 -34744.919} C_VEL
LIN {X 0,Y 101.379,Z 568.899,A -85,B 0,C 180,E1 -34746.086,E2 -34746.086} C_VEL
LIN {X 0,Y 102.611,Z 567.231,A -85,B 0,C 180,E1 -34749.437,E2 -34749.437} C_VEL
LIN {X 0,Y 103.424,Z 566.196,A -85,B 0,C 180,E1 -34750.541,E2 -34750.541} C_VEL
LIN {X 0,Y 104.543,Z 564.758,A -85,B 0,C 180,E1 -34751.597,E2 -34751.597} C_VEL
LIN {X 0,Y 105.972,Z 563.038,A -85,B 0,C 180,E1 -34753.377,E2 -34753.377} C_VEL
LIN {X 0,Y 107.161,Z 561.858,A -85,B 0,C 180,E1 -34755.158,E2 -34755.158} C_VEL
LIN {X 0,Y 110.178,Z 558.28,A -85,B 0,C 180,E1 -34757.522,E2 -34757.522} C_VEL
LIN {X 0,Y 111.448,Z 556.705,A -85,B 0,C 180,E1 -34758.316,E2 -34758.316} C_VEL
LIN {X 0,Y 112.935,Z 555.397,A -85,B 0,C 180,E1 -34759.946,E2 -34759.946} C_VEL
LIN {X 0,Y 115.864,Z 552.167,A -85,B 0,C 180,E1 -34761.97,E2 -34761.97} C_VEL
LIN {X 0,Y 118.82,Z 548.501,A -85,B 0,C 180,E1 -34763.468,E2 -34763.468} C_VEL
LIN {X 0,Y 120.25,Z 546.542,A -85,B 0,C 180,E1 -34764.064,E2 -34764.064} C_VEL
LIN {X 0,Y 123.55,Z 543.108,A -85,B 0,C 180,E1 -34766.065,E2 -34766.065} C_VEL
LIN {X 0,Y 127.376,Z 538.365,A -85,B 0,C 180,E1 -34767.866,E2 -34767.866} C_VEL
LIN {X 0,Y 131.601,Z 532.065,A -85,B 0,C 180,E1 -34769.318,E2 -34769.318} C_VEL
LIN {X 0,Y 135.553,Z 524.885,A -85,B 0,C 180,E1 -34770.346,E2 -34770.346} C_VEL
LIN {X 0,Y 140.495,Z 517.799,A -85,B 0,C 180,E1 -34772.399,E2 -34772.399} C_VEL
LIN {X 0,Y 144.379,Z 510.693,A -85,B 0,C 180,E1 -34773.704,E2 -34773.704} C_VEL
LIN {X 0,Y 149.236,Z 499.257,A -85,B 0,C 180,E1 -34775.175,E2 -34775.175} C_VEL
LIN {X 0,Y 149.45,Z 498.959,A -85,B 0,C 180,E1 -34775.276,E2 -34775.276} C_VEL
LIN {X 0,Y 147.536,Z 512.923,A -85,B 0,C 180,E1 -34776.188,E2 -34776.188} C_VEL
LIN {X 0,Y 144.617,Z 526.549,A -85,B 0,C 180,E1 -34777.444,E2 -34777.444} C_VEL
LIN {X 0,Y 140.713,Z 539.379,A -85,B 0,C 180,E1 -34778.942,E2 -34778.942} C_VEL
LIN {X 0,Y 135.83,Z 552.335,A -85,B 0,C 180,E1 -34781.047,E2 -34781.047} C_VEL
LIN {X 0,Y 130.49,Z 564.053,A -85,B 0,C 180,E1 -34783.56,E2 -34783.56} C_VEL
LIN {X 0,Y 124.672,Z 574.785,A -85,B 0,C 180,E1 -34786.509,E2 -34786.509} C_VEL
LIN {X 0,Y 117.986,Z 585.404,A -85,B 0,C 180,E1 -34790.343,E2 -34790.343} C_VEL
LIN {X 0,Y 111.856,Z 594.168,A -85,B 0,C 180,E1 -34794.603,E2 -34794.603} C_VEL
LIN {X 0,Y 106.367,Z 601.463,A -85,B 0,C 180,E1 -34799.313,E2 -34799.313} C_VEL
LIN {X 0,Y 100.66,Z 608.47,A -85,B 0,C 180,E1 -34805.323,E2 -34805.323} C_VEL
LIN {X 0,Y 95.617,Z 614.757,A -85,B 0,C 180,E1 -34812.962,E2 -34812.962} C_VEL
LIN {X 0,Y 92.17,Z 619.455,A -85,B 0,C 180,E1 -34821.258,E2 -34821.258} C_VEL
LIN {X 0,Y 90.569,Z 622.696,A -85,B 0,C 180,E1 -34830.001,E2 -34830.001} C_VEL
LIN {X 0,Y 90.703,Z 624.598,A -85,B 0,C 180,E1 -34838.885,E2 -34838.885} C_VEL
LIN {X 0,Y 92.571,Z 625.218,A -85,B 0,C 180,E1 -34847.618,E2 -34847.618} C_VEL
LIN {X 0,Y 96.178,Z 624.549,A -85,B 0,C 180,E1 -34855.911,E2 -34855.911} C_VEL
LIN {X 0,Y 101.693,Z 622.533,A -85,B 0,C 180,E1 -34863.438,E2 -34863.438} C_VEL
LIN {X 0,Y 108.5,Z 619.152,A -85,B 0,C 180,E1 -34870.209,E2 -34870.209} C_VEL
LIN {X 0,Y 116.489,Z 614.284,A -85,B 0,C 180,E1 -34876.184,E2 -34876.184} C_VEL
LIN {X 0,Y 123.152,Z 609.541,A -85,B 0,C 180,E1 -34880.161,E2 -34880.161} C_VEL
LIN {X 0,Y 131.473,Z 602.686,A -85,B 0,C 180,E1 -34884.339,E2 -34884.339} C_VEL
LIN {X 0,Y 140.42,Z 594.14,A -85,B 0,C 180,E1 -34887.995,E2 -34887.995} C_VEL
LIN {X 0,Y 148.304,Z 585.358,A -85,B 0,C 180,E1 -34890.732,E2 -34890.732} C_VEL
LIN {X 0,Y 148.546,Z 584.63,A -85,B 0,C 180,E1 -34891.246,E2 -34891.246} C_VEL
LIN {X 0,Y 138.429,Z 590.303,A -85,B 0,C 180,E1 -34894.524,E2 -34894.524} C_VEL
LIN {X 0,Y 126.218,Z 596.549,A -85,B 0,C 180,E1 -34900.635,E2 -34900.635} C_VEL
LIN {X 0,Y 118.508,Z 600.623,A -85,B 0,C 180,E1 -34906.324,E2 -34906.324} C_VEL
LIN {X 0,Y 115.076,Z 602.697,A -85,B 0,C 180,E1 -34909.478,E2 -34909.478} C_VEL
LIN {X 0,Y 106.67,Z 609.619,A -85,B 0,C 180,E1 -34923.764,E2 -34923.764} C_VEL
LIN {X 0,Y 105.643,Z 612.64,A -85,B 0,C 180,E1 -34931.472,E2 -34931.472} C_VEL
LIN {X 0,Y 110.538,Z 617.759,A -85,B 0,C 180,E1 -34946.331,E2 -34946.331} C_VEL
LIN {X 0,Y 115.964,Z 619.977,A -85,B 0,C 180,E1 -34952.929,E2 -34952.929} C_VEL
LIN {X 0,Y 123.172,Z 621.868,A -85,B 0,C 180,E1 -34958.721,E2 -34958.721} C_VEL
LIN {X 0,Y 123.962,Z 622.873,A -85,B 0,C 180,E1 -34960.134,E2 -34960.134} C_VEL
LIN {X 0,Y 115.9,Z 628.582,A -85,B 0,C 180,E1 -34963.511,E2 -34963.511} C_VEL
LIN {X 0,Y 108.914,Z 633.209,A -85,B 0,C 180,E1 -34967.524,E2 -34967.524} C_VEL
LIN {X 0,Y 100.941,Z 638.047,A -85,B 0,C 180,E1 -34973.854,E2 -34973.854} C_VEL
LIN {X 0,Y 96.119,Z 640.697,A -85,B 0,C 180,E1 -34979.328,E2 -34979.328} C_VEL
LIN {X 0,Y 91.495,Z 643.112,A -85,B 0,C 180,E1 -34987.493,E2 -34987.493} C_VEL
LIN {X 0,Y 89.319,Z 644.261,A -85,B 0,C 180,E1 -34996.392,E2 -34996.392} C_VEL
LIN {X 0,Y 89.883,Z 644.174,A -85,B 0,C 180,E1 -35005.53,E2 -35005.53} C_VEL
LIN {X 0,Y 93.108,Z 642.841,A -85,B 0,C 180,E1 -35014.314,E2 -35014.314} C_VEL
LIN {X 0,Y 98.962,Z 640.252,A -85,B 0,C 180,E1 -35022.259,E2 -35022.259} C_VEL
LIN {X 0,Y 104.943,Z 637.034,A -85,B 0,C 180,E1 -35028.042,E2 -35028.042} C_VEL
LIN {X 0,Y 106.319,Z 636.419,A -85,B 0,C 180,E1 -35029.232,E2 -35029.232} C_VEL
LIN {X 0,Y 107.755,Z 646.183,A -85,B 0,C 180,E1 -35035.922,E2 -35035.922} C_VEL
LIN {X 0,Y 112.162,Z 657.215,A -85,B 0,C 180,E1 -35044.197,E2 -35044.197} C_VEL
LIN {X 0,Y 120.221,Z 667.659,A -85,B 0,C 180,E1 -35052.068,E2 -35052.068} C_VEL
LIN {X 0,Y 124.163,Z 671.368,A -85,B 0,C 180,E1 -35054.821,E2 -35054.821} C_VEL
LIN {X 0,Y 122.268,Z 669.604,A -85,B 0,C 180,E1 -35056.572,E2 -35056.572} C_VEL
LIN {X 0,Y 114.327,Z 660.517,A -85,B 0,C 180,E1 -35063.276,E2 -35063.276} C_VEL
LIN {X 0,Y 108.81,Z 649.989,A -85,B 0,C 180,E1 -35071.133,E2 -35071.133} C_VEL
LIN {X 0,Y 106.334,Z 639.195,A -85,B 0,C 180,E1 -35078.76,E2 -35078.76} C_VEL
LIN {X 0,Y 105.695,Z 631.313,A -85,B 0,C 180,E1 -35083.546,E2 -35083.546} C_VEL
LIN {X 0,Y 104.862,Z 624.874,A -85,B 0,C 180,E1 -35086.481,E2 -35086.481} C_VEL
LIN {X 0,Y 103.507,Z 613.333,A -85,B 0,C 180,E1 -35090.752,E2 -35090.752} C_VEL
LIN {X 0,Y 102.908,Z 606.992,A -85,B 0,C 180,E1 -35092.755,E2 -35092.755} C_VEL
LIN {X 0,Y 102.107,Z 603.43,A -85,B 0,C 180,E1 -35093.53,E2 -35093.53} C_VEL
LIN {X 0,Y 99.579,Z 597.35,A -85,B 0,C 180,E1 -35094.036,E2 -35094.036} C_VEL
LIN {X 0,Y 97.008,Z 591.035,A -85,B 0,C 180,E1 -35094.424,E2 -35094.424} C_VEL
LIN {X 0,Y 96.251,Z 587.149,A -85,B 0,C 180,E1 -35095.031,E2 -35095.031} C_VEL
LIN {X 0,Y 95.688,Z 578.75,A -85,B 0,C 180,E1 -35096.854,E2 -35096.854} C_VEL
LIN {X 0,Y 94.628,Z 579.655,A -85,B 0,C 180,E1 -35097.88,E2 -35097.88} C_VEL
LIN {X 0,Y 94.268,Z 579.444,A -85,B 0,C 180,E1 -35100.001,E2 -35100.001} C_VEL
LIN {X 0,Y 95.35,Z 577.642,A -85,B 0,C 180,E1 -35102.106,E2 -35102.106} C_VEL
LIN {X 0,Y 96.255,Z 575.974,A -85,B 0,C 180,E1 -35106.268,E2 -35106.268} C_VEL
LIN {X 0,Y 97.759,Z 573.957,A -85,B 0,C 180,E1 -35108.24,E2 -35108.24} C_VEL
LIN {X 0,Y 99.779,Z 571.726,A -85,B 0,C 180,E1 -35112.159,E2 -35112.159} C_VEL
LIN {X 0,Y 102.1,Z 569.171,A -85,B 0,C 180,E1 -35114.477,E2 -35114.477} C_VEL
LIN {X 0,Y 104.17,Z 567.233,A -85,B 0,C 180,E1 -35117.08,E2 -35117.08} C_VEL
LIN {X 0,Y 107.935,Z 563.368,A -85,B 0,C 180,E1 -35119.921,E2 -35119.921} C_VEL
LIN {X 0,Y 109.19,Z 561.992,A -85,B 0,C 180,E1 -35120.661,E2 -35120.661} C_VEL
LIN {X 0,Y 110.96,Z 560.507,A -85,B 0,C 180,E1 -35122.258,E2 -35122.258} C_VEL
LIN {X 0,Y 115.75,Z 555.733,A -85,B 0,C 180,E1 -35125.063,E2 -35125.063} C_VEL
LIN {X 0,Y 119.933,Z 550.873,A -85,B 0,C 180,E1 -35126.819,E2 -35126.819} C_VEL
LIN {X 0,Y 124.131,Z 546.754,A -85,B 0,C 180,E1 -35128.982,E2 -35128.982} C_VEL
LIN {X 0,Y 129.411,Z 540.529,A -85,B 0,C 180,E1 -35130.946,E2 -35130.946} C_VEL
LIN {X 0,Y 134.424,Z 533.231,A -85,B 0,C 180,E1 -35132.284,E2 -35132.284} C_VEL
LIN {X 0,Y 137.176,Z 528.566,A -85,B 0,C 180,E1 -35132.857,E2 -35132.857} C_VEL
LIN {X 0,Y 141.673,Z 522.635,A -85,B 0,C 180,E1 -35134.484,E2 -35134.484} C_VEL
LIN {X 0,Y 141.664,Z 523.431,A -85,B 0,C 180,E1 -35134.695,E2 -35134.695} C_VEL
LIN {X 0,Y 137.943,Z 536.271,A -85,B 0,C 180,E1 -35136.064,E2 -35136.064} C_VEL
LIN {X 0,Y 133.229,Z 549.117,A -85,B 0,C 180,E1 -35137.944,E2 -35137.944} C_VEL
LIN {X 0,Y 127.635,Z 561.608,A -85,B 0,C 180,E1 -35140.409,E2 -35140.409} C_VEL
LIN {X 0,Y 121.462,Z 572.926,A -85,B 0,C 180,E1 -35143.277,E2 -35143.277} C_VEL
LIN {X 0,Y 114.941,Z 583.2,A -85,B 0,C 180,E1 -35146.72,E2 -35146.72} C_VEL
LIN {X 0,Y 108.192,Z 592.628,A -85,B 0,C 180,E1 -35150.978,E2 -35150.978} C_VEL
LIN {X 0,Y 101.322,Z 601.331,A -85,B 0,C 180,E1 -35156.425,E2 -35156.425} C_VEL
LIN {X 0,Y 95.911,Z 607.599,A -85,B 0,C 180,E1 -35161.661,E2 -35161.661} C_VEL
LIN {X 0,Y 91.404,Z 612.736,A -85,B 0,C 180,E1 -35167.471,E2 -35167.471} C_VEL
LIN {X 0,Y 86.835,Z 618.172,A -85,B 0,C 180,E1 -35175.997,E2 -35175.997} C_VEL
LIN {X 0,Y 84.125,Z 622.09,A -85,B 0,C 180,E1 -35185.225,E2 -35185.225} C_VEL
LIN {X 0,Y 83.353,Z 624.617,A -85,B 0,C 180,E1 -35194.821,E2 -35194.821} C_VEL
LIN {X 0,Y 84.542,Z 625.845,A -85,B 0,C 180,E1 -35204.393,E2 -35204.393} C_VEL
LIN {X 0,Y 87.602,Z 625.796,A -85,B 0,C 180,E1 -35213.566,E2 -35213.566} C_VEL
LIN {X 0,Y 92.67,Z 624.426,A -85,B 0,C 180,E1 -35221.945,E2 -35221.945} C_VEL
LIN {X 0,Y 99.345,Z 621.711,A -85,B 0,C 180,E1 -35229.388,E2 -35229.388} C_VEL
LIN {X 0,Y 107.296,Z 617.572,A -85,B 0,C 180,E1 -35235.898,E2 -35235.898} C_VEL
LIN {X 0,Y 116.298,Z 611.875,A -85,B 0,C 180,E1 -35241.534,E2 -35241.534} C_VEL
LIN {X 0,Y 124.054,Z 606.073,A -85,B 0,C 180,E1 -35245.433,E2 -35245.433} C_VEL
LIN {X 0,Y 132.731,Z 598.586,A -85,B 0,C 180,E1 -35249.043,E2 -35249.043} C_VEL
LIN {X 0,Y 136.781,Z 594.667,A -85,B 0,C 180,E1 -35250.524,E2 -35250.524} C_VEL
LIN {X 0,Y 138.089,Z 592.928,A -85,B 0,C 180,E1 -35251.499,E2 -35251.499} C_VEL
LIN {X 0,Y 133.375,Z 595.202,A -85,B 0,C 180,E1 -35253.227,E2 -35253.227} C_VEL
LIN {X 0,Y 120.63,Z 601.143,A -85,B 0,C 180,E1 -35259.61,E2 -35259.61} C_VEL
LIN {X 0,Y 109.048,Z 607.027,A -85,B 0,C 180,E1 -35268.889,E2 -35268.889} C_VEL
LIN {X 0,Y 100.449,Z 613.626,A -85,B 0,C 180,E1 -35283.998,E2 -35283.998} C_VEL
LIN {X 0,Y 99.574,Z 616.462,A -85,B 0,C 180,E1 -35292.182,E2 -35292.182} C_VEL
LIN {X 0,Y 104.983,Z 621.403,A -85,B 0,C 180,E1 -35307.841,E2 -35307.841} C_VEL
LIN {X 0,Y 111.155,Z 623.615,A -85,B 0,C 180,E1 -35314.994,E2 -35314.994} C_VEL
LIN {X 0,Y 114.464,Z 624.433,A -85,B 0,C 180,E1 -35317.728,E2 -35317.728} C_VEL
LIN {X 0,Y 115.227,Z 625.247,A -85,B 0,C 180,E1 -35319.113,E2 -35319.113} C_VEL
LIN {X 0,Y 106.138,Z 631.106,A -85,B 0,C 180,E1 -35323.453,E2 -35323.453} C_VEL
LIN {X 0,Y 97.282,Z 636.267,A -85,B 0,C 180,E1 -35329.607,E2 -35329.607} C_VEL
LIN {X 0,Y 90.082,Z 639.987,A -85,B 0,C 180,E1 -35337.023,E2 -35337.023} C_VEL
LIN {X 0,Y 84.957,Z 642.372,A -85,B 0,C 180,E1 -35345.654,E2 -35345.654} C_VEL
LIN {X 0,Y 82.375,Z 643.49,A -85,B 0,C 180,E1 -35355.22,E2 -35355.22} C_VEL
LIN {X 0,Y 82.722,Z 643.372,A -85,B 0,C 180,E1 -35365.142,E2 -35365.142} C_VEL
LIN {X 0,Y 85.924,Z 642.008,A -85,B 0,C 180,E1 -35374.675,E2 -35374.675} C_VEL
LIN {X 0,Y 91.886,Z 639.385,A -85,B 0,C 180,E1 -35383.219,E2 -35383.219} C_VEL
LIN {X 0,Y 97.601,Z 636.46,A -85,B 0,C 180,E1 -35388.841,E2 -35388.841} C_VEL
LIN {X 0,Y 101.667,Z 634.243,A -85,B 0,C 180,E1 -35392.263,E2 -35392.263} C_VEL
LIN {X 0,Y 103.695,Z 644.122,A -85,B 0,C 180,E1 -35399.322,E2 -35399.322} C_VEL
LIN {X 0,Y 108.212,Z 653.927,A -85,B 0,C 180,E1 -35406.779,E2 -35406.779} C_VEL
LIN {X 0,Y 115.892,Z 663.648,A -85,B 0,C 180,E1 -35414.031,E2 -35414.031} C_VEL
LIN {X 0,Y 116.69,Z 664.444,A -85,B 0,C 180,E1 -35415.48,E2 -35415.48} C_VEL
LIN {X 0,Y 108.219,Z 653.908,A -85,B 0,C 180,E1 -35423.224,E2 -35423.224} C_VEL
LIN {X 0,Y 103.545,Z 643.948,A -85,B 0,C 180,E1 -35430.632,E2 -35430.632} C_VEL
LIN {X 0,Y 101.372,Z 633.947,A -85,B 0,C 180,E1 -35437.666,E2 -35437.666} C_VEL
LIN {X 0,Y 100.644,Z 626.972,A -85,B 0,C 180,E1 -35441.912,E2 -35441.912} C_VEL
LIN {X 0,Y 99.294,Z 618.091,A -85,B 0,C 180,E1 -35445.707,E2 -35445.707} C_VEL
LIN {X 0,Y 97.885,Z 606.854,A -85,B 0,C 180,E1 -35449.696,E2 -35449.696} C_VEL
LIN {X 0,Y 96.538,Z 592.394,A -85,B 0,C 180,E1 -35453.753,E2 -35453.753} C_VEL
LIN {X 0,Y 96.251,Z 587.149,A -85,B 0,C 180,E1 -35455.031,E2 -35455.031} C_VEL
LIN {X 0,Y 95.838,Z 584.501,A -85,B 0,C 180,E1 -35456.077,E2 -35456.077} C_VEL
LIN {X 0,Y 95.023,Z 582.141,A -85,B 0,C 180,E1 -35458.098,E2 -35458.098} C_VEL
LIN {X 0,Y 93.967,Z 580.401,A -85,B 0,C 180,E1 -35461.454,E2 -35461.454} C_VEL
LIN {X 0,Y 93.522,Z 579.341,A -85,B 0,C 180,E1 -35467.962,E2 -35467.962} C_VEL
LIN {X 0,Y 94.676,Z 578.231,A -85,B 0,C 180,E1 -35471.768,E2 -35471.768} C_VEL
LIN {X 0,Y 95.38,Z 577.561,A -85,B 0,C 180,E1 -35472.922,E2 -35472.922} C_VEL
LIN {X 0,Y 97.004,Z 576.065,A -85,B 0,C 180,E1 -35475.039,E2 -35475.039} C_VEL
LIN {X 0,Y 98.625,Z 574.507,A -85,B 0,C 180,E1 -35476.505,E2 -35476.505} C_VEL
LIN {X 0,Y 103.311,Z 570.45,A -85,B 0,C 180,E1 -35480.957,E2 -35480.957} C_VEL
LIN {X 0,Y 106.937,Z 567.053,A -85,B 0,C 180,E1 -35483.143,E2 -35483.143} C_VEL
LIN {X 0,Y 110.157,Z 564.433,A -85,B 0,C 180,E1 -35485.418,E2 -35485.418} C_VEL
LIN {X 0,Y 115.161,Z 559.849,A -85,B 0,C 180,E1 -35487.913,E2 -35487.913} C_VEL
LIN {X 0,Y 119.993,Z 554.92,A -85,B 0,C 180,E1 -35489.751,E2 -35489.751} C_VEL
LIN {X 0,Y 125.43,Z 549.784,A -85,B 0,C 180,E1 -35492.041,E2 -35492.041} C_VEL
LIN {X 0,Y 129.562,Z 545.247,A -85,B 0,C 180,E1 -35493.342,E2 -35493.342} C_VEL
LIN {X 0,Y 131.86,Z 542.431,A -85,B 0,C 180,E1 -35493.931,E2 -35493.931} C_VEL
